LIN {X 0,Y 257.253,Z 513.083,A -85,B 0,C 180,E1 -18787.513,E2 -18787.513} C_VEL
LIN {X 0,Y 254.562,Z 521.781,A -85,B 0,C 180,E1 -18789.728,E2 -18789.728} C_VEL
LIN {X 0,Y 252.293,Z 529.293,A -85,B 0,C 180,E1 -18792.156,E2 -18792.156} C_VEL
LIN {X 0,Y 250.394,Z 535.119,A -85,B 0,C 180,E1 -18794.535,E2 -18794.535} C_VEL
LIN {X 0,Y 248.86,Z 539.729,A -85,B 0,C 180,E1 -18796.942,E2 -18796.942} C_VEL
LIN {X 0,Y 247.896,Z 543.258,A -85,B 0,C 180,E1 -18799.38,E2 -18799.38} C_VEL
LIN {X 0,Y 247.266,Z 545.801,A -85,B 0,C 180,E1 -18801.829,E2 -18801.829} C_VEL
LIN {X 0,Y 247.011,Z 547.002,A -85,B 0,C 180,E1 -18803.465,E2 -18803.465} C_VEL
LIN {X 0,Y 246.916,Z 548.152,A -85,B 0,C 180,E1 -18806.736,E2 -18806.736} C_VEL
LIN {X 0,Y 246.997,Z 548.151,A -85,B 0,C 180,E1 -18808.369,E2 -18808.369} C_VEL
LIN {X 0,Y 247.028,Z 547.759,A -85,B 0,C 180,E1 -18809.999,E2 -18809.999} C_VEL
LIN {X 0,Y 247.02,Z 546.926,A -85,B 0,C 180,E1 -18811.63,E2 -18811.63} C_VEL
LIN {X 0,Y 246.98,Z 545.678,A -85,B 0,C 180,E1 -18813.262,E2 -18813.262} C_VEL
LIN {X 0,Y 246.984,Z 543.722,A -85,B 0,C 180,E1 -18815.163,E2 -18815.163} C_VEL
LIN {X 0,Y 247.156,Z 540.666,A -85,B 0,C 180,E1 -18817.351,E2 -18817.351} C_VEL
LIN {X 0,Y 247.53,Z 536.217,A -85,B 0,C 180,E1 -18819.808,E2 -18819.808} C_VEL
LIN {X 0,Y 248.187,Z 530.545,A -85,B 0,C 180,E1 -18822.261,E2 -18822.261} C_VEL
LIN {X 0,Y 249.393,Z 523.451,A -85,B 0,C 180,E1 -18824.691,E2 -18824.691} C_VEL
LIN {X 0,Y 250.655,Z 516.203,A -85,B 0,C 180,E1 -18826.701,E2 -18826.701} C_VEL
LIN {X 0,Y 252.124,Z 506.524,A -85,B 0,C 180,E1 -18828.879,E2 -18828.879} C_VEL
LIN {X 0,Y 253.731,Z 496.53,A -85,B 0,C 180,E1 -18830.68,E2 -18830.68} C_VEL
LIN {X 0,Y 255.423,Z 485.697,A -85,B 0,C 180,E1 -18832.23,E2 -18832.23} C_VEL
LIN {X 0,Y 257.066,Z 473.51,A -85,B 0,C 180,E1 -18833.567,E2 -18833.567} C_VEL
LIN {X 0,Y 258.522,Z 460.783,A -85,B 0,C 180,E1 -18834.599,E2 -18834.599} C_VEL
LIN {X 0,Y 259.525,Z 448.241,A -85,B 0,C 180,E1 -18835.299,E2 -18835.299} C_VEL
LIN {X 0,Y 260.096,Z 431.393,A -85,B 0,C 180,E1 -18835.851,E2 -18835.851} C_VEL
LIN {X 0,Y 261.403,Z 385.497,A -85,B 0,C 180,E1 -18837.079,E2 -18837.079} C_VEL
LIN {X 0,Y 257.137,Z 350.583,A -85,B 0,C 180,E1 -18838.529,E2 -18838.529} C_VEL
LIN {X 0,Y 256.159,Z 345.324,A -85,B 0,C 180,E1 -18838.787,E2 -18838.787} C_VEL
LIN {X 0,Y 252.427,Z 335.153,A -85,B 0,C 180,E1 -18839.536,E2 -18839.536} C_VEL
LIN {X 0,Y 250.251,Z 324.745,A -85,B 0,C 180,E1 -18843.339,E2 -18843.339} C_VEL
LIN {X 0,Y 249.089,Z 319.458,A -85,B 0,C 180,E1 -18845.38,E2 -18845.38} C_VEL
LIN {X 0,Y 249.027,Z 319.467,A -85,B 0,C 180,E1 -18848.379,E2 -18848.379} C_VEL
LIN {X 0,Y 249,Z 319.469,A -85,B 0,C 180,E1 -18852.79,E2 -18852.79} C_VEL
LIN {X 0,Y 249.008,Z 319.467,A -85,B 0,C 180,E1 -18857.361,E2 -18857.361} C_VEL
LIN {X 0,Y 249.024,Z 319.466,A -85,B 0,C 180,E1 -18861.618,E2 -18861.618} C_VEL
LIN {X 0,Y 249.041,Z 319.463,A -85,B 0,C 180,E1 -18865.639,E2 -18865.639} C_VEL
LIN {X 0,Y 249.049,Z 319.463,A -85,B 0,C 180,E1 -18869.472,E2 -18869.472} C_VEL
LIN {X 0,Y 249.07,Z 319.462,A -85,B 0,C 180,E1 -18873.161,E2 -18873.161} C_VEL
LIN {X 0,Y 249.076,Z 319.46,A -85,B 0,C 180,E1 -18876.732,E2 -18876.732} C_VEL
LIN {X 0,Y 249.108,Z 319.453,A -85,B 0,C 180,E1 -18880.211,E2 -18880.211} C_VEL
LIN {X 0,Y 249.239,Z 319.439,A -85,B 0,C 180,E1 -18883.621,E2 -18883.621} C_VEL
LIN {X 0,Y 249.249,Z 319.422,A -85,B 0,C 180,E1 -18888.616,E2 -18888.616} C_VEL
LIN {X 0,Y 249.476,Z 319.408,A -85,B 0,C 180,E1 -18891.902,E2 -18891.902} C_VEL
LIN {X 0,Y 249.43,Z 319.409,A -85,B 0,C 180,E1 -18896.769,E2 -18896.769} C_VEL
LIN {X 0,Y 249.717,Z 319.366,A -85,B 0,C 180,E1 -18900,E2 -18900} C_VEL
LIN {X 0,Y 249.428,Z 319.412,A -85,B 0,C 180,E1 -18903.23,E2 -18903.23} C_VEL
LIN {X 0,Y 249.428,Z 319.41,A -85,B 0,C 180,E1 -18906.548,E2 -18906.548} C_VEL
LIN {X 0,Y 249.339,Z 319.412,A -85,B 0,C 180,E1 -18909.736,E2 -18909.736} C_VEL
LIN {X 0,Y 249.201,Z 319.442,A -85,B 0,C 180,E1 -18914.703,E2 -18914.703} C_VEL
LIN {X 0,Y 249.134,Z 319.446,A -85,B 0,C 180,E1 -18918.077,E2 -18918.077} C_VEL
LIN {X 0,Y 249.08,Z 319.446,A -85,B 0,C 180,E1 -18921.518,E2 -18921.518} C_VEL
LIN {X 0,Y 249.113,Z 319.452,A -85,B 0,C 180,E1 -18925.476,E2 -18925.476} C_VEL
LIN {X 0,Y 249.079,Z 319.446,A -85,B 0,C 180,E1 -18928.994,E2 -18928.994} C_VEL
LIN {X 0,Y 249.027,Z 319.459,A -85,B 0,C 180,E1 -18932.426,E2 -18932.426} C_VEL
LIN {X 0,Y 249.043,Z 319.461,A -85,B 0,C 180,E1 -18936.343,E2 -18936.343} C_VEL
LIN {X 0,Y 249.002,Z 319.461,A -85,B 0,C 180,E1 -18940.478,E2 -18940.478} C_VEL
LIN {X 0,Y 248.998,Z 319.469,A -85,B 0,C 180,E1 -18942.791,E2 -18942.791} C_VEL
LIN {X 0,Y 248.977,Z 319.469,A -85,B 0,C 180,E1 -18947.356,E2 -18947.356} C_VEL
LIN {X 0,Y 249.038,Z 319.457,A -85,B 0,C 180,E1 -18952.201,E2 -18952.201} C_VEL
LIN {X 0,Y 249.04,Z 319.463,A -85,B 0,C 180,E1 -18955.64,E2 -18955.64} C_VEL
LIN {X 0,Y 248.991,Z 319.466,A -85,B 0,C 180,E1 -18959.466,E2 -18959.466} C_VEL
LIN {X 0,Y 249.014,Z 319.463,A -85,B 0,C 180,E1 -18963.156,E2 -18963.156} C_VEL
LIN {X 0,Y 249.018,Z 319.465,A -85,B 0,C 180,E1 -18966.727,E2 -18966.727} C_VEL
LIN {X 0,Y 249.107,Z 319.48,A -85,B 0,C 180,E1 -18970.25,E2 -18970.25} C_VEL
LIN {X 0,Y 250.158,Z 322.4,A -85,B 0,C 180,E1 -18970.459,E2 -18970.459} C_VEL
LIN {X 0,Y 254.562,Z 332.022,A -85,B 0,C 180,E1 -18971.233,E2 -18971.233} C_VEL
LIN {X 0,Y 261.497,Z 350.837,A -85,B 0,C 180,E1 -18972.499,E2 -18972.499} C_VEL
LIN {X 0,Y 262.283,Z 353.529,A -85,B 0,C 180,E1 -18972.654,E2 -18972.654} C_VEL
LIN {X 0,Y 260.108,Z 426.14,A -85,B 0,C 180,E1 -18974.626,E2 -18974.626} C_VEL
LIN {X 0,Y 259.371,Z 439.258,A -85,B 0,C 180,E1 -18975.285,E2 -18975.285} C_VEL
LIN {X 0,Y 258.324,Z 451.887,A -85,B 0,C 180,E1 -18976.229,E2 -18976.229} C_VEL
LIN {X 0,Y 257.112,Z 463.144,A -85,B 0,C 180,E1 -18977.369,E2 -18977.369} C_VEL
LIN {X 0,Y 255.161,Z 474.833,A -85,B 0,C 180,E1 -18978.884,E2 -18978.884} C_VEL
LIN {X 0,Y 253.619,Z 485.254,A -85,B 0,C 180,E1 -18980.631,E2 -18980.631} C_VEL
LIN {X 0,Y 252.118,Z 493.801,A -85,B 0,C 180,E1 -18982.392,E2 -18982.392} C_VEL
LIN {X 0,Y 250.826,Z 501.662,A -85,B 0,C 180,E1 -18984.373,E2 -18984.373} C_VEL
LIN {X 0,Y 249.426,Z 509.37,A -85,B 0,C 180,E1 -18986.77,E2 -18986.77} C_VEL
LIN {X 0,Y 248.464,Z 515.541,A -85,B 0,C 180,E1 -18989.19,E2 -18989.19} C_VEL
LIN {X 0,Y 247.694,Z 520.458,A -85,B 0,C 180,E1 -18991.626,E2 -18991.626} C_VEL
LIN {X 0,Y 247.377,Z 524.246,A -85,B 0,C 180,E1 -18994.073,E2 -18994.073} C_VEL
LIN {X 0,Y 247.112,Z 527.029,A -85,B 0,C 180,E1 -18996.533,E2 -18996.533} C_VEL
LIN {X 0,Y 246.903,Z 528.355,A -85,B 0,C 180,E1 -18998.183,E2 -18998.183} C_VEL
LIN {X 0,Y 246.8,Z 529.286,A -85,B 0,C 180,E1 -18999.838,E2 -18999.838} C_VEL
LIN {X 0,Y 246.83,Z 529.798,A -85,B 0,C 180,E1 -19001.497,E2 -19001.497} C_VEL
LIN {X 0,Y 247.025,Z 529.882,A -85,B 0,C 180,E1 -19003.157,E2 -19003.157} C_VEL
LIN {X 0,Y 247.338,Z 529.537,A -85,B 0,C 180,E1 -19004.964,E2 -19004.964} C_VEL
LIN {X 0,Y 247.629,Z 528.884,A -85,B 0,C 180,E1 -19006.488,E2 -19006.488} C_VEL
LIN {X 0,Y 248.082,Z 527.744,A -85,B 0,C 180,E1 -19008.158,E2 -19008.158} C_VEL
LIN {X 0,Y 249.053,Z 525.234,A -85,B 0,C 180,E1 -19010.655,E2 -19010.655} C_VEL
LIN {X 0,Y 250.39,Z 521.674,A -85,B 0,C 180,E1 -19013.139,E2 -19013.139} C_VEL
LIN {X 0,Y 252.11,Z 516.953,A -85,B 0,C 180,E1 -19015.601,E2 -19015.601} C_VEL
LIN {X 0,Y 254.147,Z 510.919,A -85,B 0,C 180,E1 -19018.041,E2 -19018.041} C_VEL
LIN {X 0,Y 256.653,Z 503.353,A -85,B 0,C 180,E1 -19020.437,E2 -19020.437} C_VEL
LIN {X 0,Y 259.061,Z 495.585,A -85,B 0,C 180,E1 -19022.398,E2 -19022.398} C_VEL
LIN {X 0,Y 261.749,Z 486.067,A -85,B 0,C 180,E1 -19024.323,E2 -19024.323} C_VEL
LIN {X 0,Y 264.345,Z 475.395,A -85,B 0,C 180,E1 -19026.032,E2 -19026.032} C_VEL
LIN {X 0,Y 266.477,Z 465.074,A -85,B 0,C 180,E1 -19027.344,E2 -19027.344} C_VEL
LIN {X 0,Y 268.474,Z 453.071,A -85,B 0,C 180,E1 -19028.536,E2 -19028.536} C_VEL
LIN {X 0,Y 269.983,Z 440.573,A -85,B 0,C 180,E1 -19029.444,E2 -19029.444} C_VEL
LIN {X 0,Y 270.997,Z 428.372,A -85,B 0,C 180,E1 -19030.052,E2 -19030.052} C_VEL
LIN {X 0,Y 272.213,Z 404.536,A -85,B 0,C 180,E1 -19030.702,E2 -19030.702} C_VEL
LIN {X 0,Y 273.903,Z 366.243,A -85,B 0,C 180,E1 -19031.667,E2 -19031.667} C_VEL
LIN {X 0,Y 267.043,Z 351.29,A -85,B 0,C 180,E1 -19033.238,E2 -19033.238} C_VEL
LIN {X 0,Y 260.131,Z 338.414,A -85,B 0,C 180,E1 -19034.869,E2 -19034.869} C_VEL
LIN {X 0,Y 253.898,Z 327.876,A -85,B 0,C 180,E1 -19036.414,E2 -19036.414} C_VEL
LIN {X 0,Y 251.287,Z 323.854,A -85,B 0,C 180,E1 -19037.081,E2 -19037.081} C_VEL
LIN {X 0,Y 249.658,Z 321.603,A -85,B 0,C 180,E1 -19037.499,E2 -19037.499} C_VEL
LIN {X 0,Y 249.109,Z 319.866,A -85,B 0,C 180,E1 -19037.725,E2 -19037.725} C_VEL
LIN {X 0,Y 249.017,Z 319.466,A -85,B 0,C 180,E1 -19038.047,E2 -19038.047} C_VEL
LIN {X 0,Y 249.043,Z 319.458,A -85,B 0,C 180,E1 -19042.201,E2 -19042.201} C_VEL
LIN {X 0,Y 249.044,Z 319.457,A -85,B 0,C 180,E1 -19045.64,E2 -19045.64} C_VEL
LIN {X 0,Y 249.052,Z 319.447,A -85,B 0,C 180,E1 -19049.474,E2 -19049.474} C_VEL
LIN {X 0,Y 249.07,Z 319.445,A -85,B 0,C 180,E1 -19053.162,E2 -19053.162} C_VEL
LIN {X 0,Y 249.062,Z 319.446,A -85,B 0,C 180,E1 -19056.731,E2 -19056.731} C_VEL
LIN {X 0,Y 249.108,Z 319.442,A -85,B 0,C 180,E1 -19060.212,E2 -19060.212} C_VEL
LIN {X 0,Y 249.243,Z 319.433,A -85,B 0,C 180,E1 -19063.622,E2 -19063.622} C_VEL
LIN {X 0,Y 249.254,Z 319.428,A -85,B 0,C 180,E1 -19068.617,E2 -19068.617} C_VEL
LIN {X 0,Y 249.485,Z 319.406,A -85,B 0,C 180,E1 -19071.903,E2 -19071.903} C_VEL
LIN {X 0,Y 249.436,Z 319.409,A -85,B 0,C 180,E1 -19076.77,E2 -19076.77} C_VEL
LIN {X 0,Y 249.722,Z 319.376,A -85,B 0,C 180,E1 -19080,E2 -19080} C_VEL
LIN {X 0,Y 249.643,Z 319.378,A -85,B 0,C 180,E1 -19081.777,E2 -19081.777} C_VEL
LIN {X 0,Y 248.799,Z 319.482,A -85,B 0,C 180,E1 -19083.121,E2 -19083.121} C_VEL
LIN {X 0,Y 245.894,Z 319.852,A -85,B 0,C 180,E1 -19085.314,E2 -19085.314} C_VEL
LIN {X 0,Y 243.517,Z 320.143,A -85,B 0,C 180,E1 -19087.099,E2 -19087.099} C_VEL
LIN {X 0,Y 242.483,Z 320.272,A -85,B 0,C 180,E1 -19088.482,E2 -19088.482} C_VEL
LIN {X 0,Y 242.384,Z 320.284,A -85,B 0,C 180,E1 -19088.951,E2 -19088.951} C_VEL
LIN {X 0,Y 242.168,Z 320.316,A -85,B 0,C 180,E1 -19093.425,E2 -19093.425} C_VEL
LIN {X 0,Y 242.152,Z 320.311,A -85,B 0,C 180,E1 -19096.872,E2 -19096.872} C_VEL
LIN {X 0,Y 242.028,Z 320.333,A -85,B 0,C 180,E1 -19101.687,E2 -19101.687} C_VEL
LIN {X 0,Y 242.069,Z 320.328,A -85,B 0,C 180,E1 -19105.838,E2 -19105.838} C_VEL
LIN {X 0,Y 242.009,Z 320.334,A -85,B 0,C 180,E1 -19109.583,E2 -19109.583} C_VEL
LIN {X 0,Y 241.983,Z 320.338,A -85,B 0,C 180,E1 -19113.493,E2 -19113.493} C_VEL
LIN {X 0,Y 241.989,Z 320.341,A -85,B 0,C 180,E1 -19117.582,E2 -19117.582} C_VEL
LIN {X 0,Y 241.932,Z 320.329,A -85,B 0,C 180,E1 -19121.924,E2 -19121.924} C_VEL
LIN {X 0,Y 241.986,Z 320.464,A -85,B 0,C 180,E1 -19125.087,E2 -19125.087} C_VEL
LIN {X 0,Y 244.554,Z 329.275,A -85,B 0,C 180,E1 -19129.602,E2 -19129.602} C_VEL
LIN {X 0,Y 245.765,Z 333.657,A -85,B 0,C 180,E1 -19131.684,E2 -19131.684} C_VEL
LIN {X 0,Y 248.353,Z 338.358,A -85,B 0,C 180,E1 -19132.407,E2 -19132.407} C_VEL
LIN {X 0,Y 256.334,Z 353.521,A -85,B 0,C 180,E1 -19134.512,E2 -19134.512} C_VEL
LIN {X 0,Y 262.927,Z 367.737,A -85,B 0,C 180,E1 -19136.166,E2 -19136.166} C_VEL
LIN {X 0,Y 264.065,Z 371.108,A -85,B 0,C 180,E1 -19136.47,E2 -19136.47} C_VEL
LIN {X 0,Y 267.144,Z 390.198,A -85,B 0,C 180,E1 -19137.602,E2 -19137.602} C_VEL
LIN {X 0,Y 264.881,Z 443.227,A -85,B 0,C 180,E1 -19139.029,E2 -19139.029} C_VEL
LIN {X 0,Y 263.521,Z 456.86,A -85,B 0,C 180,E1 -19139.665,E2 -19139.665} C_VEL
LIN {X 0,Y 261.592,Z 469.409,A -85,B 0,C 180,E1 -19140.528,E2 -19140.528} C_VEL
LIN {X 0,Y 259.274,Z 481.377,A -85,B 0,C 180,E1 -19141.682,E2 -19141.682} C_VEL
LIN {X 0,Y 256.566,Z 492.822,A -85,B 0,C 180,E1 -19143.129,E2 -19143.129} C_VEL
LIN {X 0,Y 253.805,Z 503.151,A -85,B 0,C 180,E1 -19144.802,E2 -19144.802} C_VEL
LIN {X 0,Y 251.249,Z 511.614,A -85,B 0,C 180,E1 -19146.509,E2 -19146.509} C_VEL
LIN {X 0,Y 248.707,Z 519.442,A -85,B 0,C 180,E1 -19148.447,E2 -19148.447} C_VEL
LIN {X 0,Y 246.267,Z 527.109,A -85,B 0,C 180,E1 -19150.841,E2 -19150.841} C_VEL
LIN {X 0,Y 244.208,Z 533.294,A -85,B 0,C 180,E1 -19153.274,E2 -19153.274} C_VEL
LIN {X 0,Y 242.408,Z 538.231,A -85,B 0,C 180,E1 -19155.733,E2 -19155.733} C_VEL
LIN {X 0,Y 241.211,Z 542.064,A -85,B 0,C 180,E1 -19158.231,E2 -19158.231} C_VEL
LIN {X 0,Y 240.216,Z 545.635,A -85,B 0,C 180,E1 -19161.588,E2 -19161.588} C_VEL
LIN {X 0,Y 239.953,Z 546.795,A -85,B 0,C 180,E1 -19163.271,E2 -19163.271} C_VEL
LIN {X 0,Y 239.816,Z 547.898,A -85,B 0,C 180,E1 -19166.639,E2 -19166.639} C_VEL
LIN {X 0,Y 239.903,Z 547.876,A -85,B 0,C 180,E1 -19168.321,E2 -19168.321} C_VEL
LIN {X 0,Y 239.957,Z 547.451,A -85,B 0,C 180,E1 -19169.999,E2 -19169.999} C_VEL
LIN {X 0,Y 239.927,Z 546.584,A -85,B 0,C 180,E1 -19171.678,E2 -19171.678} C_VEL
LIN {X 0,Y 239.879,Z 545.313,A -85,B 0,C 180,E1 -19173.359,E2 -19173.359} C_VEL
LIN {X 0,Y 239.919,Z 542.599,A -85,B 0,C 180,E1 -19175.884,E2 -19175.884} C_VEL
LIN {X 0,Y 240.178,Z 538.844,A -85,B 0,C 180,E1 -19178.412,E2 -19178.412} C_VEL
LIN {X 0,Y 240.703,Z 533.946,A -85,B 0,C 180,E1 -19180.94,E2 -19180.94} C_VEL
LIN {X 0,Y 241.585,Z 527.758,A -85,B 0,C 180,E1 -19183.457,E2 -19183.457} C_VEL
LIN {X 0,Y 242.909,Z 520.055,A -85,B 0,C 180,E1 -19185.953,E2 -19185.953} C_VEL
LIN {X 0,Y 244.376,Z 512.158,A -85,B 0,C 180,E1 -19188.008,E2 -19188.008} C_VEL
LIN {X 0,Y 245.855,Z 502.462,A -85,B 0,C 180,E1 -19190.061,E2 -19190.061} C_VEL
LIN {X 0,Y 247.707,Z 491.733,A -85,B 0,C 180,E1 -19191.862,E2 -19191.862} C_VEL
LIN {X 0,Y 249.32,Z 481.357,A -85,B 0,C 180,E1 -19193.243,E2 -19193.243} C_VEL
LIN {X 0,Y 250.912,Z 468.939,A -85,B 0,C 180,E1 -19194.512,E2 -19194.512} C_VEL
LIN {X 0,Y 252.312,Z 455.866,A -85,B 0,C 180,E1 -19195.467,E2 -19195.467} C_VEL
LIN {X 0,Y 253.19,Z 443.052,A -85,B 0,C 180,E1 -19196.089,E2 -19196.089} C_VEL
LIN {X 0,Y 254.817,Z 385.79,A -85,B 0,C 180,E1 -19197.694,E2 -19197.694} C_VEL
LIN {X 0,Y 250.723,Z 351.896,A -85,B 0,C 180,E1 -19199.15,E2 -19199.15} C_VEL
LIN {X 0,Y 249.794,Z 347.296,A -85,B 0,C 180,E1 -19199.392,E2 -19199.392} C_VEL
LIN {X 0,Y 245.198,Z 334.962,A -85,B 0,C 180,E1 -19200.308,E2 -19200.308} C_VEL
LIN {X 0,Y 242.927,Z 324.358,A -85,B 0,C 180,E1 -19204.342,E2 -19204.342} C_VEL
LIN {X 0,Y 242.051,Z 320.334,A -85,B 0,C 180,E1 -19206.01,E2 -19206.01} C_VEL
LIN {X 0,Y 241.956,Z 320.346,A -85,B 0,C 180,E1 -19209.718,E2 -19209.718} C_VEL
LIN {X 0,Y 241.917,Z 320.352,A -85,B 0,C 180,E1 -19214.204,E2 -19214.204} C_VEL
LIN {X 0,Y 241.932,Z 320.349,A -85,B 0,C 180,E1 -19218.076,E2 -19218.076} C_VEL
LIN {X 0,Y 241.984,Z 320.344,A -85,B 0,C 180,E1 -19222.417,E2 -19222.417} C_VEL
LIN {X 0,Y 241.978,Z 320.345,A -85,B 0,C 180,E1 -19226.507,E2 -19226.507} C_VEL
LIN {X 0,Y 242.034,Z 320.339,A -85,B 0,C 180,E1 -19230.586,E2 -19230.586} C_VEL
LIN {X 0,Y 242.065,Z 320.331,A -85,B 0,C 180,E1 -19234.182,E2 -19234.182} C_VEL
LIN {X 0,Y 242.05,Z 320.331,A -85,B 0,C 180,E1 -19238.296,E2 -19238.296} C_VEL
LIN {X 0,Y 242.16,Z 320.322,A -85,B 0,C 180,E1 -19243.278,E2 -19243.278} C_VEL
LIN {X 0,Y 242.183,Z 320.301,A -85,B 0,C 180,E1 -19248.279,E2 -19248.279} C_VEL
LIN {X 0,Y 242.423,Z 320.284,A -85,B 0,C 180,E1 -19251.665,E2 -19251.665} C_VEL
LIN {X 0,Y 242.254,Z 320.307,A -85,B 0,C 180,E1 -19255.007,E2 -19255.007} C_VEL
LIN {X 0,Y 242.632,Z 320.246,A -85,B 0,C 180,E1 -19258.34,E2 -19258.34} C_VEL
LIN {X 0,Y 242.631,Z 320.254,A -85,B 0,C 180,E1 -19261.659,E2 -19261.659} C_VEL
LIN {X 0,Y 242.404,Z 320.285,A -85,B 0,C 180,E1 -19266.659,E2 -19266.659} C_VEL
LIN {X 0,Y 242.263,Z 320.292,A -85,B 0,C 180,E1 -19270.024,E2 -19270.024} C_VEL
LIN {X 0,Y 242.163,Z 320.318,A -85,B 0,C 180,E1 -19275.141,E2 -19275.141} C_VEL
LIN {X 0,Y 242.067,Z 320.321,A -85,B 0,C 180,E1 -19278.624,E2 -19278.624} C_VEL
LIN {X 0,Y 242.002,Z 320.331,A -85,B 0,C 180,E1 -19282.181,E2 -19282.181} C_VEL
LIN {X 0,Y 242.063,Z 320.331,A -85,B 0,C 180,E1 -19285.838,E2 -19285.838} C_VEL
LIN {X 0,Y 242.026,Z 320.323,A -85,B 0,C 180,E1 -19289.58,E2 -19289.58} C_VEL
LIN {X 0,Y 241.977,Z 320.34,A -85,B 0,C 180,E1 -19293.493,E2 -19293.493} C_VEL
LIN {X 0,Y 241.985,Z 320.332,A -85,B 0,C 180,E1 -19297.582,E2 -19297.582} C_VEL
LIN {X 0,Y 241.93,Z 320.346,A -85,B 0,C 180,E1 -19301.924,E2 -19301.924} C_VEL
LIN {X 0,Y 241.901,Z 320.342,A -85,B 0,C 180,E1 -19306.579,E2 -19306.579} C_VEL
LIN {X 0,Y 241.99,Z 320.335,A -85,B 0,C 180,E1 -19311.642,E2 -19311.642} C_VEL
LIN {X 0,Y 241.984,Z 320.341,A -85,B 0,C 180,E1 -19314.49,E2 -19314.49} C_VEL
LIN {X 0,Y 241.945,Z 320.345,A -85,B 0,C 180,E1 -19318.477,E2 -19318.477} C_VEL
LIN {X 0,Y 241.95,Z 320.342,A -85,B 0,C 180,E1 -19322.306,E2 -19322.306} C_VEL
LIN {X 0,Y 241.991,Z 320.341,A -85,B 0,C 180,E1 -19326.01,E2 -19326.01} C_VEL
LIN {X 0,Y 242.018,Z 320.339,A -85,B 0,C 180,E1 -19329.426,E2 -19329.426} C_VEL
LIN {X 0,Y 243.035,Z 323.201,A -85,B 0,C 180,E1 -19329.669,E2 -19329.669} C_VEL
LIN {X 0,Y 247.68,Z 332.843,A -85,B 0,C 180,E1 -19330.512,E2 -19330.512} C_VEL
LIN {X 0,Y 254.536,Z 350.896,A -85,B 0,C 180,E1 -19331.808,E2 -19331.808} C_VEL
LIN {X 0,Y 255.778,Z 354.774,A -85,B 0,C 180,E1 -19332.052,E2 -19332.052} C_VEL
LIN {X 0,Y 253.504,Z 426.848,A -85,B 0,C 180,E1 -19334.06,E2 -19334.06} C_VEL
LIN {X 0,Y 252.689,Z 440.569,A -85,B 0,C 180,E1 -19334.783,E2 -19334.783} C_VEL
LIN {X 0,Y 251.612,Z 452.915,A -85,B 0,C 180,E1 -19335.751,E2 -19335.751} C_VEL
LIN {X 0,Y 250.262,Z 464.743,A -85,B 0,C 180,E1 -19337.018,E2 -19337.018} C_VEL
LIN {X 0,Y 248.442,Z 474.903,A -85,B 0,C 180,E1 -19338.373,E2 -19338.373} C_VEL
LIN {X 0,Y 246.826,Z 485.36,A -85,B 0,C 180,E1 -19340.164,E2 -19340.164} C_VEL
LIN {X 0,Y 245.114,Z 494.815,A -85,B 0,C 180,E1 -19342.173,E2 -19342.173} C_VEL
LIN {X 0,Y 243.538,Z 503.893,A -85,B 0,C 180,E1 -19344.619,E2 -19344.619} C_VEL
LIN {X 0,Y 242.134,Z 511.228,A -85,B 0,C 180,E1 -19347.089,E2 -19347.089} C_VEL
LIN {X 0,Y 241.11,Z 517.947,A -85,B 0,C 180,E1 -19350.001,E2 -19350.001} C_VEL
LIN {X 0,Y 240.426,Z 522.397,A -85,B 0,C 180,E1 -19352.514,E2 -19352.514} C_VEL
LIN {X 0,Y 240.18,Z 525.767,A -85,B 0,C 180,E1 -19355.037,E2 -19355.037} C_VEL
LIN {X 0,Y 239.982,Z 527.454,A -85,B 0,C 180,E1 -19356.728,E2 -19356.728} C_VEL
LIN {X 0,Y 239.792,Z 528.744,A -85,B 0,C 180,E1 -19358.427,E2 -19358.427} C_VEL
LIN {X 0,Y 239.723,Z 529.635,A -85,B 0,C 180,E1 -19360.132,E2 -19360.132} C_VEL
LIN {X 0,Y 239.776,Z 530.083,A -85,B 0,C 180,E1 -19361.84,E2 -19361.84} C_VEL
LIN {X 0,Y 240.309,Z 529.794,A -85,B 0,C 180,E1 -19365.261,E2 -19365.261} C_VEL
LIN {X 0,Y 240.648,Z 529.054,A -85,B 0,C 180,E1 -19366.981,E2 -19366.981} C_VEL
LIN {X 0,Y 241.152,Z 527.856,A -85,B 0,C 180,E1 -19368.698,E2 -19368.698} C_VEL
LIN {X 0,Y 241.845,Z 526.242,A -85,B 0,C 180,E1 -19370.409,E2 -19370.409} C_VEL
LIN {X 0,Y 243.163,Z 522.965,A -85,B 0,C 180,E1 -19372.966,E2 -19372.966} C_VEL
LIN {X 0,Y 244.862,Z 518.568,A -85,B 0,C 180,E1 -19375.501,E2 -19375.501} C_VEL
LIN {X 0,Y 247.006,Z 512.67,A -85,B 0,C 180,E1 -19378.112,E2 -19378.112} C_VEL
LIN {X 0,Y 249.444,Z 505.79,A -85,B 0,C 180,E1 -19380.474,E2 -19380.474} C_VEL
LIN {X 0,Y 252.406,Z 496.805,A -85,B 0,C 180,E1 -19382.886,E2 -19382.886} C_VEL
LIN {X 0,Y 255.171,Z 487.541,A -85,B 0,C 180,E1 -19384.855,E2 -19384.855} C_VEL
LIN {X 0,Y 257.856,Z 477.179,A -85,B 0,C 180,E1 -19386.6,E2 -19386.6} C_VEL
LIN {X 0,Y 260.392,Z 465.583,A -85,B 0,C 180,E1 -19388.127,E2 -19388.127} C_VEL
LIN {X 0,Y 262.492,Z 453.54,A -85,B 0,C 180,E1 -19389.349,E2 -19389.349} C_VEL
LIN {X 0,Y 264.13,Z 440.525,A -85,B 0,C 180,E1 -19390.309,E2 -19390.309} C_VEL
LIN {X 0,Y 265.185,Z 428.167,A -85,B 0,C 180,E1 -19390.928,E2 -19390.928} C_VEL
LIN {X 0,Y 266.582,Z 400.796,A -85,B 0,C 180,E1 -19391.674,E2 -19391.674} C_VEL
LIN {X 0,Y 268.012,Z 368.143,A -85,B 0,C 180,E1 -19392.521,E2 -19392.521} C_VEL
LIN {X 0,Y 260.943,Z 352.931,A -85,B 0,C 180,E1 -19394.219,E2 -19394.219} C_VEL
LIN {X 0,Y 254.159,Z 340.365,A -85,B 0,C 180,E1 -19395.906,E2 -19395.906} C_VEL
LIN {X 0,Y 249.492,Z 332.557,A -85,B 0,C 180,E1 -19397.116,E2 -19397.116} C_VEL
LIN {X 0,Y 246.884,Z 328.628,A -85,B 0,C 180,E1 -19397.807,E2 -19397.807} C_VEL
LIN {X 0,Y 244.466,Z 324.912,A -85,B 0,C 180,E1 -19398.471,E2 -19398.471} C_VEL
LIN {X 0,Y 242.615,Z 322.568,A -85,B 0,C 180,E1 -19398.974,E2 -19398.974} C_VEL
LIN {X 0,Y 241.977,Z 320.342,A -85,B 0,C 180,E1 -19399.252,E2 -19399.252} C_VEL
LIN {X 0,Y 241.989,Z 320.338,A -85,B 0,C 180,E1 -19402.418,E2 -19402.418} C_VEL
LIN {X 0,Y 241.981,Z 320.334,A -85,B 0,C 180,E1 -19406.508,E2 -19406.508} C_VEL
LIN {X 0,Y 242.037,Z 320.327,A -85,B 0,C 180,E1 -19410.588,E2 -19410.588} C_VEL
LIN {X 0,Y 242.068,Z 320.325,A -85,B 0,C 180,E1 -19414.183,E2 -19414.183} C_VEL
LIN {X 0,Y 242.027,Z 320.333,A -85,B 0,C 180,E1 -19418.314,E2 -19418.314} C_VEL
LIN {X 0,Y 242.164,Z 320.318,A -85,B 0,C 180,E1 -19423.279,E2 -19423.279} C_VEL
LIN {X 0,Y 242.187,Z 320.31,A -85,B 0,C 180,E1 -19428.28,E2 -19428.28} C_VEL
LIN {X 0,Y 242.436,Z 320.286,A -85,B 0,C 180,E1 -19431.666,E2 -19431.666} C_VEL
LIN {X 0,Y 242.26,Z 320.304,A -85,B 0,C 180,E1 -19435.008,E2 -19435.008} C_VEL
LIN {X 0,Y 242.637,Z 320.249,A -85,B 0,C 180,E1 -19438.341,E2 -19438.341} C_VEL
LIN {X 0,Y 242.629,Z 320.252,A -85,B 0,C 180,E1 -19441.694,E2 -19441.694} C_VEL
LIN {X 0,Y 242.434,Z 320.272,A -85,B 0,C 180,E1 -19446.659,E2 -19446.659} C_VEL
LIN {X 0,Y 242.384,Z 320.284,A -85,B 0,C 180,E1 -19448.951,E2 -19448.951} C_VEL
LIN {X 0,Y 241.655,Z 320.381,A -85,B 0,C 180,E1 -19450.336,E2 -19450.336} C_VEL
LIN {X 0,Y 238.711,Z 320.744,A -85,B 0,C 180,E1 -19452.593,E2 -19452.593} C_VEL
LIN {X 0,Y 236.236,Z 321.055,A -85,B 0,C 180,E1 -19454.431,E2 -19454.431} C_VEL
LIN {X 0,Y 235.176,Z 321.178,A -85,B 0,C 180,E1 -19455.861,E2 -19455.861} C_VEL
LIN {X 0,Y 235.09,Z 321.188,A -85,B 0,C 180,E1 -19456.345,E2 -19456.345} C_VEL
LIN {X 0,Y 235,Z 321.202,A -85,B 0,C 180,E1 -19461.032,E2 -19461.032} C_VEL
LIN {X 0,Y 234.996,Z 321.211,A -85,B 0,C 180,E1 -19466.206,E2 -19466.206} C_VEL
LIN {X 0,Y 234.924,Z 321.223,A -85,B 0,C 180,E1 -19470.569,E2 -19470.569} C_VEL
LIN {X 0,Y 234.929,Z 321.219,A -85,B 0,C 180,E1 -19474.639,E2 -19474.639} C_VEL
LIN {X 0,Y 234.915,Z 321.204,A -85,B 0,C 180,E1 -19478.936,E2 -19478.936} C_VEL
LIN {X 0,Y 234.899,Z 321.306,A -85,B 0,C 180,E1 -19483.661,E2 -19483.661} C_VEL
LIN {X 0,Y 237.521,Z 330.019,A -85,B 0,C 180,E1 -19488.403,E2 -19488.403} C_VEL
LIN {X 0,Y 238.489,Z 333.51,A -85,B 0,C 180,E1 -19490.066,E2 -19490.066} C_VEL
LIN {X 0,Y 240.919,Z 337.776,A -85,B 0,C 180,E1 -19490.795,E2 -19490.795} C_VEL
LIN {X 0,Y 245.507,Z 345.979,A -85,B 0,C 180,E1 -19492.111,E2 -19492.111} C_VEL
LIN {X 0,Y 251.873,Z 358.247,A -85,B 0,C 180,E1 -19493.847,E2 -19493.847} C_VEL
LIN {X 0,Y 257.799,Z 371.218,A -85,B 0,C 180,E1 -19495.401,E2 -19495.401} C_VEL
LIN {X 0,Y 258.724,Z 374.033,A -85,B 0,C 180,E1 -19495.662,E2 -19495.662} C_VEL
LIN {X 0,Y 261.44,Z 391.461,A -85,B 0,C 180,E1 -19496.723,E2 -19496.723} C_VEL
LIN {X 0,Y 259.081,Z 443.047,A -85,B 0,C 180,E1 -19498.129,E2 -19498.129} C_VEL
LIN {X 0,Y 257.65,Z 456.817,A -85,B 0,C 180,E1 -19498.783,E2 -19498.783} C_VEL
LIN {X 0,Y 255.68,Z 469.299,A -85,B 0,C 180,E1 -19499.663,E2 -19499.663} C_VEL
LIN {X 0,Y 253.436,Z 480.433,A -85,B 0,C 180,E1 -19500.741,E2 -19500.741} C_VEL
LIN {X 0,Y 250.666,Z 491.995,A -85,B 0,C 180,E1 -19502.217,E2 -19502.217} C_VEL
LIN {X 0,Y 247.732,Z 502.422,A -85,B 0,C 180,E1 -19503.913,E2 -19503.913} C_VEL
LIN {X 0,Y 244.775,Z 511.84,A -85,B 0,C 180,E1 -19505.848,E2 -19505.848} C_VEL
LIN {X 0,Y 241.629,Z 520.932,A -85,B 0,C 180,E1 -19508.232,E2 -19508.232} C_VEL
LIN {X 0,Y 239.156,Z 528.287,A -85,B 0,C 180,E1 -19510.699,E2 -19510.699} C_VEL
LIN {X 0,Y 236.708,Z 535.061,A -85,B 0,C 180,E1 -19513.616,E2 -19513.616} C_VEL
LIN {X 0,Y 234.984,Z 539.561,A -85,B 0,C 180,E1 -19516.156,E2 -19516.156} C_VEL
LIN {X 0,Y 234.246,Z 541.948,A -85,B 0,C 180,E1 -19517.876,E2 -19517.876} C_VEL
LIN {X 0,Y 233.185,Z 545.47,A -85,B 0,C 180,E1 -19521.332,E2 -19521.332} C_VEL
LIN {X 0,Y 232.732,Z 547.305,A -85,B 0,C 180,E1 -19524.802,E2 -19524.802} C_VEL
LIN {X 0,Y 232.811,Z 547.6,A -85,B 0,C 180,E1 -19528.27,E2 -19528.27} C_VEL
LIN {X 0,Y 232.888,Z 547.133,A -85,B 0,C 180,E1 -19529.999,E2 -19529.999} C_VEL
LIN {X 0,Y 232.836,Z 546.241,A -85,B 0,C 180,E1 -19531.729,E2 -19531.729} C_VEL
LIN {X 0,Y 232.778,Z 543.541,A -85,B 0,C 180,E1 -19534.905,E2 -19534.905} C_VEL
LIN {X 0,Y 233.021,Z 539.789,A -85,B 0,C 180,E1 -19537.8,E2 -19537.8} C_VEL
LIN {X 0,Y 233.468,Z 535.234,A -85,B 0,C 180,E1 -19540.405,E2 -19540.405} C_VEL
LIN {X 0,Y 234.435,Z 528.304,A -85,B 0,C 180,E1 -19543.434,E2 -19543.434} C_VEL
LIN {X 0,Y 235.808,Z 520.783,A -85,B 0,C 180,E1 -19546.002,E2 -19546.002} C_VEL
LIN {X 0,Y 237.413,Z 512.293,A -85,B 0,C 180,E1 -19548.326,E2 -19548.326} C_VEL
LIN {X 0,Y 238.944,Z 502.665,A -85,B 0,C 180,E1 -19550.442,E2 -19550.442} C_VEL
LIN {X 0,Y 240.86,Z 492.034,A -85,B 0,C 180,E1 -19552.291,E2 -19552.291} C_VEL
LIN {X 0,Y 242.762,Z 480.153,A -85,B 0,C 180,E1 -19553.909,E2 -19553.909} C_VEL
LIN {X 0,Y 244.443,Z 467.387,A -85,B 0,C 180,E1 -19555.205,E2 -19555.205} C_VEL
LIN {X 0,Y 245.783,Z 454.621,A -85,B 0,C 180,E1 -19556.137,E2 -19556.137} C_VEL
LIN {X 0,Y 246.617,Z 442.388,A -85,B 0,C 180,E1 -19556.725,E2 -19556.725} C_VEL
LIN {X 0,Y 248.324,Z 386.94,A -85,B 0,C 180,E1 -19558.309,E2 -19558.309} C_VEL
LIN {X 0,Y 244.568,Z 354.753,A -85,B 0,C 180,E1 -19559.728,E2 -19559.728} C_VEL
LIN {X 0,Y 243.673,Z 349.917,A -85,B 0,C 180,E1 -19559.984,E2 -19559.984} C_VEL
LIN {X 0,Y 237.879,Z 334.594,A -85,B 0,C 180,E1 -19561.205,E2 -19561.205} C_VEL
LIN {X 0,Y 235.526,Z 323.603,A -85,B 0,C 180,E1 -19565.564,E2 -19565.564} C_VEL
LIN {X 0,Y 234.998,Z 321.213,A -85,B 0,C 180,E1 -19566.552,E2 -19566.552} C_VEL
LIN {X 0,Y 234.88,Z 321.227,A -85,B 0,C 180,E1 -19571.167,E2 -19571.167} C_VEL
LIN {X 0,Y 234.883,Z 321.227,A -85,B 0,C 180,E1 -19575.897,E2 -19575.897} C_VEL
LIN {X 0,Y 234.88,Z 321.229,A -85,B 0,C 180,E1 -19578.831,E2 -19578.831} C_VEL
LIN {X 0,Y 234.916,Z 321.225,A -85,B 0,C 180,E1 -19581.078,E2 -19581.078} C_VEL
LIN {X 0,Y 234.925,Z 321.223,A -85,B 0,C 180,E1 -19585.361,E2 -19585.361} C_VEL
LIN {X 0,Y 234.929,Z 321.223,A -85,B 0,C 180,E1 -19589.431,E2 -19589.431} C_VEL
LIN {X 0,Y 234.992,Z 321.213,A -85,B 0,C 180,E1 -19593.793,E2 -19593.793} C_VEL
LIN {X 0,Y 235.009,Z 321.211,A -85,B 0,C 180,E1 -19598.969,E2 -19598.969} C_VEL
LIN {X 0,Y 235.093,Z 321.2,A -85,B 0,C 180,E1 -19603.059,E2 -19603.059} C_VEL
LIN {X 0,Y 235.115,Z 321.182,A -85,B 0,C 180,E1 -19607.922,E2 -19607.922} C_VEL
LIN {X 0,Y 235.372,Z 321.16,A -85,B 0,C 180,E1 -19611.414,E2 -19611.414} C_VEL
LIN {X 0,Y 235.399,Z 321.161,A -85,B 0,C 180,E1 -19613.141,E2 -19613.141} C_VEL
LIN {X 0,Y 235.592,Z 321.122,A -85,B 0,C 180,E1 -19618.29,E2 -19618.29} C_VEL
LIN {X 0,Y 235.591,Z 321.131,A -85,B 0,C 180,E1 -19621.709,E2 -19621.709} C_VEL
LIN {X 0,Y 235.355,Z 321.162,A -85,B 0,C 180,E1 -19626.86,E2 -19626.86} C_VEL
LIN {X 0,Y 235.21,Z 321.17,A -85,B 0,C 180,E1 -19630.327,E2 -19630.327} C_VEL
LIN {X 0,Y 235.11,Z 321.198,A -85,B 0,C 180,E1 -19635.606,E2 -19635.606} C_VEL
LIN {X 0,Y 235.003,Z 321.198,A -85,B 0,C 180,E1 -19639.206,E2 -19639.206} C_VEL
LIN {X 0,Y 234.949,Z 321.215,A -85,B 0,C 180,E1 -19642.884,E2 -19642.884} C_VEL
LIN {X 0,Y 234.966,Z 321.214,A -85,B 0,C 180,E1 -19646.657,E2 -19646.657} C_VEL
LIN {X 0,Y 234.928,Z 321.206,A -85,B 0,C 180,E1 -19650.568,E2 -19650.568} C_VEL
LIN {X 0,Y 234.926,Z 321.222,A -85,B 0,C 180,E1 -19654.638,E2 -19654.638} C_VEL
LIN {X 0,Y 234.938,Z 321.207,A -85,B 0,C 180,E1 -19658.945,E2 -19658.945} C_VEL
LIN {X 0,Y 234.872,Z 321.224,A -85,B 0,C 180,E1 -19663.489,E2 -19663.489} C_VEL
LIN {X 0,Y 234.854,Z 321.219,A -85,B 0,C 180,E1 -19666.508,E2 -19666.508} C_VEL
LIN {X 0,Y 234.914,Z 321.218,A -85,B 0,C 180,E1 -19671.079,E2 -19671.079} C_VEL
LIN {X 0,Y 234.926,Z 321.222,A -85,B 0,C 180,E1 -19675.362,E2 -19675.362} C_VEL
LIN {X 0,Y 234.892,Z 321.221,A -85,B 0,C 180,E1 -19679.428,E2 -19679.428} C_VEL
LIN {X 0,Y 234.938,Z 321.218,A -85,B 0,C 180,E1 -19683.822,E2 -19683.822} C_VEL
LIN {X 0,Y 234.989,Z 321.214,A -85,B 0,C 180,E1 -19688.58,E2 -19688.58} C_VEL
LIN {X 0,Y 236.123,Z 324.263,A -85,B 0,C 180,E1 -19688.864,E2 -19688.864} C_VEL
LIN {X 0,Y 241.919,Z 336.28,A -85,B 0,C 180,E1 -19689.964,E2 -19689.964} C_VEL
LIN {X 0,Y 248.422,Z 353.527,A -85,B 0,C 180,E1 -19691.246,E2 -19691.246} C_VEL
LIN {X 0,Y 249.262,Z 356.427,A -85,B 0,C 180,E1 -19691.427,E2 -19691.427} C_VEL
LIN {X 0,Y 246.97,Z 426.817,A -85,B 0,C 180,E1 -19693.433,E2 -19693.433} C_VEL
LIN {X 0,Y 246.146,Z 440.37,A -85,B 0,C 180,E1 -19694.156,E2 -19694.156} C_VEL
LIN {X 0,Y 245.029,Z 452.845,A -85,B 0,C 180,E1 -19695.147,E2 -19695.147} C_VEL
LIN {X 0,Y 243.609,Z 464.767,A -85,B 0,C 180,E1 -19696.444,E2 -19696.444} C_VEL
LIN {X 0,Y 241.744,Z 474.968,A -85,B 0,C 180,E1 -19697.833,E2 -19697.833} C_VEL
LIN {X 0,Y 240.044,Z 485.462,A -85,B 0,C 180,E1 -19699.67,E2 -19699.67} C_VEL
LIN {X 0,Y 238.431,Z 494.062,A -85,B 0,C 180,E1 -19701.526,E2 -19701.526} C_VEL
LIN {X 0,Y 237.008,Z 501.97,A -85,B 0,C 180,E1 -19703.616,E2 -19703.616} C_VEL
LIN {X 0,Y 235.485,Z 509.733,A -85,B 0,C 180,E1 -19706.15,E2 -19706.15} C_VEL
LIN {X 0,Y 234.259,Z 516.841,A -85,B 0,C 180,E1 -19709.141,E2 -19709.141} C_VEL
LIN {X 0,Y 233.47,Z 521.596,A -85,B 0,C 180,E1 -19711.726,E2 -19711.726} C_VEL
LIN {X 0,Y 233.177,Z 525.231,A -85,B 0,C 180,E1 -19714.322,E2 -19714.322} C_VEL
LIN {X 0,Y 232.867,Z 527.875,A -85,B 0,C 180,E1 -19716.934,E2 -19716.934} C_VEL
LIN {X 0,Y 232.673,Z 529.133,A -85,B 0,C 180,E1 -19718.687,E2 -19718.687} C_VEL
LIN {X 0,Y 232.641,Z 529.962,A -85,B 0,C 180,E1 -19720.444,E2 -19720.444} C_VEL
LIN {X 0,Y 232.952,Z 530.385,A -85,B 0,C 180,E1 -19723.967,E2 -19723.967} C_VEL
LIN {X 0,Y 233.297,Z 530.012,A -85,B 0,C 180,E1 -19725.732,E2 -19725.732} C_VEL
LIN {X 0,Y 233.681,Z 529.205,A -85,B 0,C 180,E1 -19727.503,E2 -19727.503} C_VEL
LIN {X 0,Y 234.248,Z 527.968,A -85,B 0,C 180,E1 -19729.271,E2 -19729.271} C_VEL
LIN {X 0,Y 235.7,Z 524.675,A -85,B 0,C 180,E1 -19732.431,E2 -19732.431} C_VEL
LIN {X 0,Y 237.631,Z 520.121,A -85,B 0,C 180,E1 -19735.395,E2 -19735.395} C_VEL
LIN {X 0,Y 239.683,Z 514.795,A -85,B 0,C 180,E1 -19737.98,E2 -19737.98} C_VEL
LIN {X 0,Y 242.228,Z 508.063,A -85,B 0,C 180,E1 -19740.514,E2 -19740.514} C_VEL
LIN {X 0,Y 245.194,Z 499.653,A -85,B 0,C 180,E1 -19742.998,E2 -19742.998} C_VEL
LIN {X 0,Y 248.035,Z 490.943,A -85,B 0,C 180,E1 -19745.014,E2 -19745.014} C_VEL
LIN {X 0,Y 251.086,Z 480.12,A -85,B 0,C 180,E1 -19746.999,E2 -19746.999} C_VEL
LIN {X 0,Y 253.669,Z 469.299,A -85,B 0,C 180,E1 -19748.563,E2 -19748.563} C_VEL
LIN {X 0,Y 256.009,Z 457.264,A -85,B 0,C 180,E1 -19749.897,E2 -19749.897} C_VEL
LIN {X 0,Y 257.76,Z 445.585,A -85,B 0,C 180,E1 -19750.873,E2 -19750.873} C_VEL
LIN {X 0,Y 259.014,Z 433.206,A -85,B 0,C 180,E1 -19751.623,E2 -19751.623} C_VEL
LIN {X 0,Y 259.985,Z 420.889,A -85,B 0,C 180,E1 -19752.056,E2 -19752.056} C_VEL
LIN {X 0,Y 262.308,Z 370.35,A -85,B 0,C 180,E1 -19753.385,E2 -19753.385} C_VEL
LIN {X 0,Y 255.32,Z 355.429,A -85,B 0,C 180,E1 -19755.142,E2 -19755.142} C_VEL
LIN {X 0,Y 248.824,Z 343.462,A -85,B 0,C 180,E1 -19756.839,E2 -19756.839} C_VEL
LIN {X 0,Y 244.826,Z 336.811,A -85,B 0,C 180,E1 -19757.925,E2 -19757.925} C_VEL
LIN {X 0,Y 240.173,Z 329.858,A -85,B 0,C 180,E1 -19759.231,E2 -19759.231} C_VEL
LIN {X 0,Y 238.02,Z 326.47,A -85,B 0,C 180,E1 -19759.871,E2 -19759.871} C_VEL
LIN {X 0,Y 235.626,Z 323.56,A -85,B 0,C 180,E1 -19760.568,E2 -19760.568} C_VEL
LIN {X 0,Y 234.938,Z 321.217,A -85,B 0,C 180,E1 -19760.86,E2 -19760.86} C_VEL
LIN {X 0,Y 234.931,Z 321.214,A -85,B 0,C 180,E1 -19765.362,E2 -19765.362} C_VEL
LIN {X 0,Y 234.932,Z 321.205,A -85,B 0,C 180,E1 -19769.433,E2 -19769.433} C_VEL
LIN {X 0,Y 234.995,Z 321.202,A -85,B 0,C 180,E1 -19773.794,E2 -19773.794} C_VEL
LIN {X 0,Y 234.998,Z 321.209,A -85,B 0,C 180,E1 -19778.969,E2 -19778.969} C_VEL
LIN {X 0,Y 235.097,Z 321.201,A -85,B 0,C 180,E1 -19783.06,E2 -19783.06} C_VEL
LIN {X 0,Y 235.148,Z 321.189,A -85,B 0,C 180,E1 -19787.924,E2 -19787.924} C_VEL
LIN {X 0,Y 235.391,Z 321.164,A -85,B 0,C 180,E1 -19791.415,E2 -19791.415} C_VEL
LIN {X 0,Y 235.406,Z 321.151,A -85,B 0,C 180,E1 -19793.142,E2 -19793.142} C_VEL
LIN {X 0,Y 235.596,Z 321.126,A -85,B 0,C 180,E1 -19798.291,E2 -19798.291} C_VEL
LIN {X 0,Y 235.596,Z 321.128,A -85,B 0,C 180,E1 -19801.71,E2 -19801.71} C_VEL
LIN {X 0,Y 235.405,Z 321.147,A -85,B 0,C 180,E1 -19806.859,E2 -19806.859} C_VEL
LIN {X 0,Y 235.24,Z 321.175,A -85,B 0,C 180,E1 -19810.327,E2 -19810.327} C_VEL
LIN {X 0,Y 235.116,Z 321.186,A -85,B 0,C 180,E1 -19815.607,E2 -19815.607} C_VEL
LIN {X 0,Y 235.09,Z 321.188,A -85,B 0,C 180,E1 -19816.345,E2 -19816.345} C_VEL
LIN {X 0,Y 234.415,Z 321.282,A -85,B 0,C 180,E1 -19817.774,E2 -19817.774} C_VEL
LIN {X 0,Y 231.531,Z 321.643,A -85,B 0,C 180,E1 -19820.103,E2 -19820.103} C_VEL
LIN {X 0,Y 229.067,Z 321.95,A -85,B 0,C 180,E1 -19822.001,E2 -19822.001} C_VEL
LIN {X 0,Y 227.99,Z 322.081,A -85,B 0,C 180,E1 -19823.476,E2 -19823.476} C_VEL
LIN {X 0,Y 227.893,Z 322.089,A -85,B 0,C 180,E1 -19823.977,E2 -19823.977} C_VEL
LIN {X 0,Y 227.881,Z 322.095,A -85,B 0,C 180,E1 -19827.556,E2 -19827.556} C_VEL
LIN {X 0,Y 227.869,Z 322.094,A -85,B 0,C 180,E1 -19831.623,E2 -19831.623} C_VEL
LIN {X 0,Y 227.882,Z 322.09,A -85,B 0,C 180,E1 -19835.872,E2 -19835.872} C_VEL
LIN {X 0,Y 227.813,Z 322.077,A -85,B 0,C 180,E1 -19840.38,E2 -19840.38} C_VEL
LIN {X 0,Y 227.812,Z 322.128,A -85,B 0,C 180,E1 -19842.089,E2 -19842.089} C_VEL
LIN {X 0,Y 230.122,Z 329.673,A -85,B 0,C 180,E1 -19846.497,E2 -19846.497} C_VEL
LIN {X 0,Y 231.114,Z 333.007,A -85,B 0,C 180,E1 -19848.25,E2 -19848.25} C_VEL
LIN {X 0,Y 233.468,Z 337.184,A -85,B 0,C 180,E1 -19849.022,E2 -19849.022} C_VEL
LIN {X 0,Y 234.887,Z 339.539,A -85,B 0,C 180,E1 -19849.467,E2 -19849.467} C_VEL
LIN {X 0,Y 238.267,Z 345.316,A -85,B 0,C 180,E1 -19850.501,E2 -19850.501} C_VEL
LIN {X 0,Y 244.57,Z 357.095,A -85,B 0,C 180,E1 -19852.346,E2 -19852.346} C_VEL
LIN {X 0,Y 251.133,Z 370.982,A -85,B 0,C 180,E1 -19854.173,E2 -19854.173} C_VEL
LIN {X 0,Y 253.355,Z 376.628,A -85,B 0,C 180,E1 -19854.793,E2 -19854.793} C_VEL
LIN {X 0,Y 255.708,Z 392.306,A -85,B 0,C 180,E1 -19855.773,E2 -19855.773} C_VEL
LIN {X 0,Y 253.382,Z 442.655,A -85,B 0,C 180,E1 -19857.18,E2 -19857.18} C_VEL
LIN {X 0,Y 251.972,Z 456.036,A -85,B 0,C 180,E1 -19857.82,E2 -19857.82} C_VEL
LIN {X 0,Y 249.821,Z 469.213,A -85,B 0,C 180,E1 -19858.755,E2 -19858.755} C_VEL
LIN {X 0,Y 247.303,Z 481.085,A -85,B 0,C 180,E1 -19859.942,E2 -19859.942} C_VEL
LIN {X 0,Y 244.429,Z 492.48,A -85,B 0,C 180,E1 -19861.444,E2 -19861.444} C_VEL
LIN {X 0,Y 241.394,Z 502.776,A -85,B 0,C 180,E1 -19863.174,E2 -19863.174} C_VEL
LIN {X 0,Y 238.318,Z 512.049,A -85,B 0,C 180,E1 -19865.15,E2 -19865.15} C_VEL
LIN {X 0,Y 235.045,Z 521.054,A -85,B 0,C 180,E1 -19867.59,E2 -19867.59} C_VEL
LIN {X 0,Y 232.47,Z 528.327,A -85,B 0,C 180,E1 -19870.116,E2 -19870.116} C_VEL
LIN {X 0,Y 229.893,Z 535.023,A -85,B 0,C 180,E1 -19873.116,E2 -19873.116} C_VEL
LIN {X 0,Y 228.066,Z 539.471,A -85,B 0,C 180,E1 -19875.728,E2 -19875.728} C_VEL
LIN {X 0,Y 227.274,Z 541.833,A -85,B 0,C 180,E1 -19877.498,E2 -19877.498} C_VEL
LIN {X 0,Y 226.609,Z 543.773,A -85,B 0,C 180,E1 -19879.275,E2 -19879.275} C_VEL
LIN {X 0,Y 226.143,Z 545.295,A -85,B 0,C 180,E1 -19881.06,E2 -19881.06} C_VEL
LIN {X 0,Y 225.648,Z 547.073,A -85,B 0,C 180,E1 -19884.638,E2 -19884.638} C_VEL
LIN {X 0,Y 225.626,Z 547.389,A -85,B 0,C 180,E1 -19886.428,E2 -19886.428} C_VEL
LIN {X 0,Y 225.72,Z 547.319,A -85,B 0,C 180,E1 -19888.215,E2 -19888.215} C_VEL
LIN {X 0,Y 225.819,Z 546.813,A -85,B 0,C 180,E1 -19889.999,E2 -19889.999} C_VEL
LIN {X 0,Y 225.747,Z 545.897,A -85,B 0,C 180,E1 -19891.783,E2 -19891.783} C_VEL
LIN {X 0,Y 225.69,Z 543.408,A -85,B 0,C 180,E1 -19894.802,E2 -19894.802} C_VEL
LIN {X 0,Y 225.958,Z 539.342,A -85,B 0,C 180,E1 -19898.045,E2 -19898.045} C_VEL
LIN {X 0,Y 226.441,Z 534.728,A -85,B 0,C 180,E1 -19900.732,E2 -19900.732} C_VEL
LIN {X 0,Y 227.498,Z 527.72,A -85,B 0,C 180,E1 -19903.851,E2 -19903.851} C_VEL
LIN {X 0,Y 228.916,Z 520.128,A -85,B 0,C 180,E1 -19906.497,E2 -19906.497} C_VEL
LIN {X 0,Y 230.347,Z 513.089,A -85,B 0,C 180,E1 -19908.484,E2 -19908.484} C_VEL
LIN {X 0,Y 232.047,Z 502.868,A -85,B 0,C 180,E1 -19910.846,E2 -19910.846} C_VEL
LIN {X 0,Y 234.033,Z 492.335,A -85,B 0,C 180,E1 -19912.744,E2 -19912.744} C_VEL
LIN {X 0,Y 235.991,Z 480.613,A -85,B 0,C 180,E1 -19914.406,E2 -19914.406} C_VEL
LIN {X 0,Y 237.721,Z 468.109,A -85,B 0,C 180,E1 -19915.735,E2 -19915.735} C_VEL
LIN {X 0,Y 239.178,Z 454.919,A -85,B 0,C 180,E1 -19916.739,E2 -19916.739} C_VEL
LIN {X 0,Y 240.089,Z 441.706,A -85,B 0,C 180,E1 -19917.394,E2 -19917.394} C_VEL
LIN {X 0,Y 241.828,Z 387.017,A -85,B 0,C 180,E1 -19918.994,E2 -19918.994} C_VEL
LIN {X 0,Y 237.876,Z 353.422,A -85,B 0,C 180,E1 -19920.539,E2 -19920.539} C_VEL
LIN {X 0,Y 232.024,Z 337.968,A -85,B 0,C 180,E1 -19921.78,E2 -19921.78} C_VEL
LIN {X 0,Y 230.59,Z 334.304,A -85,B 0,C 180,E1 -19922.131,E2 -19922.131} C_VEL
LIN {X 0,Y 228.726,Z 325.581,A -85,B 0,C 180,E1 -19925.718,E2 -19925.718} C_VEL
LIN {X 0,Y 227.895,Z 322.097,A -85,B 0,C 180,E1 -19927.23,E2 -19927.23} C_VEL
LIN {X 0,Y 227.824,Z 322.108,A -85,B 0,C 180,E1 -19930.376,E2 -19930.376} C_VEL
LIN {X 0,Y 227.824,Z 322.106,A -85,B 0,C 180,E1 -19935.194,E2 -19935.194} C_VEL
LIN {X 0,Y 227.823,Z 322.106,A -85,B 0,C 180,E1 -19939.622,E2 -19939.622} C_VEL
LIN {X 0,Y 227.878,Z 322.102,A -85,B 0,C 180,E1 -19944.127,E2 -19944.127} C_VEL
LIN {X 0,Y 227.868,Z 322.101,A -85,B 0,C 180,E1 -19948.377,E2 -19948.377} C_VEL
LIN {X 0,Y 227.884,Z 322.099,A -85,B 0,C 180,E1 -19952.444,E2 -19952.444} C_VEL
LIN {X 0,Y 227.912,Z 322.095,A -85,B 0,C 180,E1 -19956.367,E2 -19956.367} C_VEL
LIN {X 0,Y 227.94,Z 322.09,A -85,B 0,C 180,E1 -19960.174,E2 -19960.174} C_VEL
LIN {X 0,Y 228.055,Z 322.076,A -85,B 0,C 180,E1 -19963.897,E2 -19963.897} C_VEL
LIN {X 0,Y 228.072,Z 322.061,A -85,B 0,C 180,E1 -19967.543,E2 -19967.543} C_VEL
LIN {X 0,Y 228.302,Z 322.038,A -85,B 0,C 180,E1 -19971.145,E2 -19971.145} C_VEL
LIN {X 0,Y 228.35,Z 322.038,A -85,B 0,C 180,E1 -19972.928,E2 -19972.928} C_VEL
LIN {X 0,Y 228.55,Z 321.999,A -85,B 0,C 180,E1 -19978.237,E2 -19978.237} C_VEL
LIN {X 0,Y 228.549,Z 322.008,A -85,B 0,C 180,E1 -19981.762,E2 -19981.762} C_VEL
LIN {X 0,Y 228.307,Z 322.04,A -85,B 0,C 180,E1 -19987.073,E2 -19987.073} C_VEL
LIN {X 0,Y 228.142,Z 322.051,A -85,B 0,C 180,E1 -19990.651,E2 -19990.651} C_VEL
LIN {X 0,Y 228.061,Z 322.078,A -85,B 0,C 180,E1 -19994.272,E2 -19994.272} C_VEL
LIN {X 0,Y 227.999,Z 322.078,A -85,B 0,C 180,E1 -19997.953,E2 -19997.953} C_VEL
LIN {X 0,Y 227.913,Z 322.085,A -85,B 0,C 180,E1 -20002.321,E2 -20002.321} C_VEL
LIN {X 0,Y 227.939,Z 322.09,A -85,B 0,C 180,E1 -20006.603,E2 -20006.603} C_VEL
LIN {X 0,Y 227.905,Z 322.079,A -85,B 0,C 180,E1 -20010.296,E2 -20010.296} C_VEL
LIN {X 0,Y 227.873,Z 322.096,A -85,B 0,C 180,E1 -20013.721,E2 -20013.721} C_VEL
LIN {X 0,Y 227.84,Z 322.092,A -85,B 0,C 180,E1 -20018.091,E2 -20018.091} C_VEL
LIN {X 0,Y 227.801,Z 322.109,A -85,B 0,C 180,E1 -20022.744,E2 -20022.744} C_VEL
LIN {X 0,Y 227.784,Z 322.105,A -85,B 0,C 180,E1 -20027.253,E2 -20027.253} C_VEL
LIN {X 0,Y 227.84,Z 322.097,A -85,B 0,C 180,E1 -20031.909,E2 -20031.909} C_VEL
LIN {X 0,Y 227.876,Z 322.098,A -85,B 0,C 180,E1 -20036.378,E2 -20036.378} C_VEL
LIN {X 0,Y 227.869,Z 322.094,A -85,B 0,C 180,E1 -20040.432,E2 -20040.432} C_VEL
LIN {X 0,Y 227.872,Z 322.097,A -85,B 0,C 180,E1 -20044.42,E2 -20044.42} C_VEL
LIN {X 0,Y 227.936,Z 322.093,A -85,B 0,C 180,E1 -20047.718,E2 -20047.718} C_VEL
LIN {X 0,Y 228.991,Z 325.036,A -85,B 0,C 180,E1 -20047.967,E2 -20047.967} C_VEL
LIN {X 0,Y 235.766,Z 338.681,A -85,B 0,C 180,E1 -20049.306,E2 -20049.306} C_VEL
LIN {X 0,Y 242.512,Z 356.664,A -85,B 0,C 180,E1 -20050.693,E2 -20050.693} C_VEL
LIN {X 0,Y 242.724,Z 360.032,A -85,B 0,C 180,E1 -20050.826,E2 -20050.826} C_VEL
LIN {X 0,Y 240.418,Z 427.524,A -85,B 0,C 180,E1 -20052.804,E2 -20052.804} C_VEL
LIN {X 0,Y 239.572,Z 440.926,A -85,B 0,C 180,E1 -20053.545,E2 -20053.545} C_VEL
LIN {X 0,Y 238.359,Z 453.836,A -85,B 0,C 180,E1 -20054.612,E2 -20054.612} C_VEL
LIN {X 0,Y 236.726,Z 466.371,A -85,B 0,C 180,E1 -20056.042,E2 -20056.042} C_VEL
LIN {X 0,Y 234.807,Z 476.328,A -85,B 0,C 180,E1 -20057.468,E2 -20057.468} C_VEL
LIN {X 0,Y 233.114,Z 486.625,A -85,B 0,C 180,E1 -20059.359,E2 -20059.359} C_VEL
LIN {X 0,Y 231.437,Z 495.078,A -85,B 0,C 180,E1 -20061.267,E2 -20061.267} C_VEL
LIN {X 0,Y 229.708,Z 504.214,A -85,B 0,C 180,E1 -20063.853,E2 -20063.853} C_VEL
LIN {X 0,Y 228.179,Z 511.585,A -85,B 0,C 180,E1 -20066.469,E2 -20066.469} C_VEL
LIN {X 0,Y 227.164,Z 517.488,A -85,B 0,C 180,E1 -20069.114,E2 -20069.114} C_VEL
LIN {X 0,Y 226.368,Z 522.163,A -85,B 0,C 180,E1 -20071.78,E2 -20071.78} C_VEL
LIN {X 0,Y 226.06,Z 525.723,A -85,B 0,C 180,E1 -20074.458,E2 -20074.458} C_VEL
LIN {X 0,Y 225.753,Z 528.297,A -85,B 0,C 180,E1 -20077.154,E2 -20077.154} C_VEL
LIN {X 0,Y 225.578,Z 529.514,A -85,B 0,C 180,E1 -20078.962,E2 -20078.962} C_VEL
LIN {X 0,Y 225.547,Z 530.281,A -85,B 0,C 180,E1 -20080.776,E2 -20080.776} C_VEL
LIN {X 0,Y 225.946,Z 530.636,A -85,B 0,C 180,E1 -20084.409,E2 -20084.409} C_VEL
LIN {X 0,Y 226.301,Z 530.218,A -85,B 0,C 180,E1 -20086.231,E2 -20086.231} C_VEL
LIN {X 0,Y 226.73,Z 529.353,A -85,B 0,C 180,E1 -20088.058,E2 -20088.058} C_VEL
LIN {X 0,Y 227.369,Z 528.081,A -85,B 0,C 180,E1 -20089.878,E2 -20089.878} C_VEL
LIN {X 0,Y 228.818,Z 525.027,A -85,B 0,C 180,E1 -20092.865,E2 -20092.865} C_VEL
LIN {X 0,Y 230.373,Z 521.554,A -85,B 0,C 180,E1 -20095.284,E2 -20095.284} C_VEL
LIN {X 0,Y 232.479,Z 516.581,A -85,B 0,C 180,E1 -20097.942,E2 -20097.942} C_VEL
LIN {X 0,Y 235.029,Z 510.274,A -85,B 0,C 180,E1 -20100.554,E2 -20100.554} C_VEL
LIN {X 0,Y 238.009,Z 502.314,A -85,B 0,C 180,E1 -20103.112,E2 -20103.112} C_VEL
LIN {X 0,Y 240.962,Z 493.864,A -85,B 0,C 180,E1 -20105.249,E2 -20105.249} C_VEL
LIN {X 0,Y 244.035,Z 484.102,A -85,B 0,C 180,E1 -20107.214,E2 -20107.214} C_VEL
LIN {X 0,Y 246.609,Z 474.162,A -85,B 0,C 180,E1 -20108.827,E2 -20108.827} C_VEL
LIN {X 0,Y 249.213,Z 462.742,A -85,B 0,C 180,E1 -20110.255,E2 -20110.255} C_VEL
LIN {X 0,Y 251.243,Z 450.662,A -85,B 0,C 180,E1 -20111.433,E2 -20111.433} C_VEL
LIN {X 0,Y 252.886,Z 437.815,A -85,B 0,C 180,E1 -20112.331,E2 -20112.331} C_VEL
LIN {X 0,Y 253.975,Z 425.342,A -85,B 0,C 180,E1 -20112.881,E2 -20112.881} C_VEL
LIN {X 0,Y 256.578,Z 372.436,A -85,B 0,C 180,E1 -20114.308,E2 -20114.308} C_VEL
LIN {X 0,Y 249.845,Z 358.093,A -85,B 0,C 180,E1 -20116.087,E2 -20116.087} C_VEL
LIN {X 0,Y 241.758,Z 343.251,A -85,B 0,C 180,E1 -20118.335,E2 -20118.335} C_VEL
LIN {X 0,Y 235.907,Z 334.622,A -85,B 0,C 180,E1 -20120.031,E2 -20120.031} C_VEL
LIN {X 0,Y 233.336,Z 330.903,A -85,B 0,C 180,E1 -20120.817,E2 -20120.817} C_VEL
LIN {X 0,Y 231.158,Z 327.508,A -85,B 0,C 180,E1 -20121.516,E2 -20121.516} C_VEL
LIN {X 0,Y 228.728,Z 324.757,A -85,B 0,C 180,E1 -20122.276,E2 -20122.276} C_VEL
LIN {X 0,Y 227.866,Z 322.096,A -85,B 0,C 180,E1 -20122.687,E2 -20122.687} C_VEL
LIN {X 0,Y 227.88,Z 322.091,A -85,B 0,C 180,E1 -20126.378,E2 -20126.378} C_VEL
LIN {X 0,Y 227.92,Z 322.085,A -85,B 0,C 180,E1 -20130.438,E2 -20130.438} C_VEL
LIN {X 0,Y 227.926,Z 322.087,A -85,B 0,C 180,E1 -20134.426,E2 -20134.426} C_VEL
LIN {X 0,Y 227.948,Z 322.087,A -85,B 0,C 180,E1 -20138.286,E2 -20138.286} C_VEL
LIN {X 0,Y 228.035,Z 322.08,A -85,B 0,C 180,E1 -20142.826,E2 -20142.826} C_VEL
LIN {X 0,Y 228.095,Z 322.07,A -85,B 0,C 180,E1 -20147.545,E2 -20147.545} C_VEL
LIN {X 0,Y 228.326,Z 322.043,A -85,B 0,C 180,E1 -20151.147,E2 -20151.147} C_VEL
LIN {X 0,Y 228.359,Z 322.03,A -85,B 0,C 180,E1 -20152.929,E2 -20152.929} C_VEL
LIN {X 0,Y 228.555,Z 322.002,A -85,B 0,C 180,E1 -20158.238,E2 -20158.238} C_VEL
LIN {X 0,Y 228.555,Z 322.004,A -85,B 0,C 180,E1 -20161.762,E2 -20161.762} C_VEL
LIN {X 0,Y 228.356,Z 322.024,A -85,B 0,C 180,E1 -20167.072,E2 -20167.072} C_VEL
LIN {X 0,Y 228.161,Z 322.054,A -85,B 0,C 180,E1 -20170.651,E2 -20170.651} C_VEL
LIN {X 0,Y 228.067,Z 322.074,A -85,B 0,C 180,E1 -20174.272,E2 -20174.272} C_VEL
LIN {X 0,Y 228.005,Z 322.081,A -85,B 0,C 180,E1 -20177.954,E2 -20177.954} C_VEL
LIN {X 0,Y 227.919,Z 322.093,A -85,B 0,C 180,E1 -20182.321,E2 -20182.321} C_VEL
LIN {X 0,Y 227.893,Z 322.089,A -85,B 0,C 180,E1 -20183.977,E2 -20183.977} C_VEL
LIN {X 0,Y 227.195,Z 322.18,A -85,B 0,C 180,E1 -20185.451,E2 -20185.451} C_VEL
LIN {X 0,Y 224.328,Z 322.535,A -85,B 0,C 180,E1 -20187.857,E2 -20187.857} C_VEL
LIN {X 0,Y 221.911,Z 322.839,A -85,B 0,C 180,E1 -20189.82,E2 -20189.82} C_VEL
LIN {X 0,Y 220.878,Z 322.968,A -85,B 0,C 180,E1 -20191.344,E2 -20191.344} C_VEL
LIN {X 0,Y 220.795,Z 322.973,A -85,B 0,C 180,E1 -20191.861,E2 -20191.861} C_VEL
LIN {X 0,Y 220.803,Z 322.975,A -85,B 0,C 180,E1 -20194.955,E2 -20194.955} C_VEL
LIN {X 0,Y 220.812,Z 322.977,A -85,B 0,C 180,E1 -20197.278,E2 -20197.278} C_VEL
LIN {X 0,Y 220.813,Z 323.151,A -85,B 0,C 180,E1 -20200.497,E2 -20200.497} C_VEL
LIN {X 0,Y 223.087,Z 330.608,A -85,B 0,C 180,E1 -20205.14,E2 -20205.14} C_VEL
LIN {X 0,Y 223.75,Z 332.643,A -85,B 0,C 180,E1 -20206.256,E2 -20206.256} C_VEL
LIN {X 0,Y 226.491,Z 337.237,A -85,B 0,C 180,E1 -20207.227,E2 -20207.227} C_VEL
LIN {X 0,Y 227.954,Z 339.667,A -85,B 0,C 180,E1 -20207.727,E2 -20207.727} C_VEL
LIN {X 0,Y 231.059,Z 344.845,A -85,B 0,C 180,E1 -20208.755,E2 -20208.755} C_VEL
LIN {X 0,Y 235.676,Z 352.841,A -85,B 0,C 180,E1 -20210.213,E2 -20210.213} C_VEL
LIN {X 0,Y 243.673,Z 368.945,A -85,B 0,C 180,E1 -20212.618,E2 -20212.618} C_VEL
LIN {X 0,Y 248.013,Z 379.096,A -85,B 0,C 180,E1 -20213.874,E2 -20213.874} C_VEL
LIN {X 0,Y 250.127,Z 393.268,A -85,B 0,C 180,E1 -20214.798,E2 -20214.798} C_VEL
LIN {X 0,Y 247.788,Z 442.025,A -85,B 0,C 180,E1 -20216.18,E2 -20216.18} C_VEL
LIN {X 0,Y 246.312,Z 455.587,A -85,B 0,C 180,E1 -20216.831,E2 -20216.831} C_VEL
LIN {X 0,Y 244.231,Z 468.021,A -85,B 0,C 180,E1 -20217.713,E2 -20217.713} C_VEL
LIN {X 0,Y 241.621,Z 480.162,A -85,B 0,C 180,E1 -20218.916,E2 -20218.916} C_VEL
LIN {X 0,Y 238.596,Z 491.68,A -85,B 0,C 180,E1 -20220.436,E2 -20220.436} C_VEL
LIN {X 0,Y 235.423,Z 502.067,A -85,B 0,C 180,E1 -20222.196,E2 -20222.196} C_VEL
LIN {X 0,Y 232.525,Z 510.575,A -85,B 0,C 180,E1 -20224.007,E2 -20224.007} C_VEL
LIN {X 0,Y 229.571,Z 518.441,A -85,B 0,C 180,E1 -20226.069,E2 -20226.069} C_VEL
LIN {X 0,Y 226.543,Z 526.395,A -85,B 0,C 180,E1 -20228.725,E2 -20228.725} C_VEL
LIN {X 0,Y 223.801,Z 533.272,A -85,B 0,C 180,E1 -20231.697,E2 -20231.697} C_VEL
LIN {X 0,Y 221.77,Z 538.042,A -85,B 0,C 180,E1 -20234.373,E2 -20234.373} C_VEL
LIN {X 0,Y 220.296,Z 541.719,A -85,B 0,C 180,E1 -20237.095,E2 -20237.095} C_VEL
LIN {X 0,Y 219.619,Z 543.635,A -85,B 0,C 180,E1 -20238.93,E2 -20238.93} C_VEL
LIN {X 0,Y 219.095,Z 545.11,A -85,B 0,C 180,E1 -20240.77,E2 -20240.77} C_VEL
LIN {X 0,Y 218.571,Z 546.842,A -85,B 0,C 180,E1 -20244.464,E2 -20244.464} C_VEL
LIN {X 0,Y 218.525,Z 547.135,A -85,B 0,C 180,E1 -20246.311,E2 -20246.311} C_VEL
LIN {X 0,Y 218.632,Z 547.028,A -85,B 0,C 180,E1 -20248.157,E2 -20248.157} C_VEL
LIN {X 0,Y 218.751,Z 546.493,A -85,B 0,C 180,E1 -20249.999,E2 -20249.999} C_VEL
LIN {X 0,Y 218.66,Z 545.553,A -85,B 0,C 180,E1 -20251.841,E2 -20251.841} C_VEL
LIN {X 0,Y 218.59,Z 543.315,A -85,B 0,C 180,E1 -20254.652,E2 -20254.652} C_VEL
LIN {X 0,Y 218.792,Z 540.162,A -85,B 0,C 180,E1 -20257.381,E2 -20257.381} C_VEL
LIN {X 0,Y 219.212,Z 535.877,A -85,B 0,C 180,E1 -20260.155,E2 -20260.155} C_VEL
LIN {X 0,Y 220.167,Z 529.365,A -85,B 0,C 180,E1 -20263.38,E2 -20263.38} C_VEL
LIN {X 0,Y 221.58,Z 522.223,A -85,B 0,C 180,E1 -20266.112,E2 -20266.112} C_VEL
LIN {X 0,Y 223.283,Z 513.842,A -85,B 0,C 180,E1 -20268.662,E2 -20268.662} C_VEL
LIN {X 0,Y 225.032,Z 504.095,A -85,B 0,C 180,E1 -20271.048,E2 -20271.048} C_VEL
LIN {X 0,Y 226.936,Z 493.93,A -85,B 0,C 180,E1 -20273.015,E2 -20273.015} C_VEL
LIN {X 0,Y 228.956,Z 482.628,A -85,B 0,C 180,E1 -20274.722,E2 -20274.722} C_VEL
LIN {X 0,Y 230.749,Z 470.924,A -85,B 0,C 180,E1 -20276.086,E2 -20276.086} C_VEL
LIN {X 0,Y 232.255,Z 459.014,A -85,B 0,C 180,E1 -20277.115,E2 -20277.115} C_VEL
LIN {X 0,Y 233.391,Z 445.947,A -85,B 0,C 180,E1 -20277.883,E2 -20277.883} C_VEL
LIN {X 0,Y 234.092,Z 427.287,A -85,B 0,C 180,E1 -20278.524,E2 -20278.524} C_VEL
LIN {X 0,Y 235.385,Z 387.668,A -85,B 0,C 180,E1 -20279.693,E2 -20279.693} C_VEL
LIN {X 0,Y 231.716,Z 355.856,A -85,B 0,C 180,E1 -20281.205,E2 -20281.205} C_VEL
LIN {X 0,Y 226.191,Z 341.079,A -85,B 0,C 180,E1 -20282.437,E2 -20282.437} C_VEL
LIN {X 0,Y 223.322,Z 334.029,A -85,B 0,C 180,E1 -20283.116,E2 -20283.116} C_VEL
LIN {X 0,Y 221.273,Z 324.751,A -85,B 0,C 180,E1 -20287.118,E2 -20287.118} C_VEL
LIN {X 0,Y 220.837,Z 322.976,A -85,B 0,C 180,E1 -20287.921,E2 -20287.921} C_VEL
LIN {X 0,Y 220.76,Z 322.987,A -85,B 0,C 180,E1 -20292.927,E2 -20292.927} C_VEL
LIN {X 0,Y 220.76,Z 322.986,A -85,B 0,C 180,E1 -20297.071,E2 -20297.071} C_VEL
LIN {X 0,Y 220.805,Z 322.983,A -85,B 0,C 180,E1 -20300.462,E2 -20300.462} C_VEL
LIN {X 0,Y 220.799,Z 322.983,A -85,B 0,C 180,E1 -20305.044,E2 -20305.044} C_VEL
LIN {X 0,Y 220.866,Z 322.975,A -85,B 0,C 180,E1 -20309.394,E2 -20309.394} C_VEL
LIN {X 0,Y 220.893,Z 322.97,A -85,B 0,C 180,E1 -20313.549,E2 -20313.549} C_VEL
LIN {X 0,Y 220.875,Z 322.97,A -85,B 0,C 180,E1 -20317.553,E2 -20317.553} C_VEL
LIN {X 0,Y 220.982,Z 322.955,A -85,B 0,C 180,E1 -20322.57,E2 -20322.57} C_VEL
LIN {X 0,Y 221.01,Z 322.943,A -85,B 0,C 180,E1 -20327.138,E2 -20327.138} C_VEL
LIN {X 0,Y 221.233,Z 322.917,A -85,B 0,C 180,E1 -20330.86,E2 -20330.86} C_VEL
LIN {X 0,Y 221.285,Z 322.918,A -85,B 0,C 180,E1 -20332.701,E2 -20332.701} C_VEL
LIN {X 0,Y 221.508,Z 322.875,A -85,B 0,C 180,E1 -20338.181,E2 -20338.181} C_VEL
LIN {X 0,Y 221.507,Z 322.885,A -85,B 0,C 180,E1 -20341.818,E2 -20341.818} C_VEL
LIN {X 0,Y 221.244,Z 322.921,A -85,B 0,C 180,E1 -20347.3,E2 -20347.3} C_VEL
LIN {X 0,Y 221.064,Z 322.934,A -85,B 0,C 180,E1 -20350.996,E2 -20350.996} C_VEL
LIN {X 0,Y 220.992,Z 322.956,A -85,B 0,C 180,E1 -20354.739,E2 -20354.739} C_VEL
LIN {X 0,Y 220.916,Z 322.954,A -85,B 0,C 180,E1 -20358.549,E2 -20358.549} C_VEL
LIN {X 0,Y 220.881,Z 322.964,A -85,B 0,C 180,E1 -20362.675,E2 -20362.675} C_VEL
LIN {X 0,Y 220.882,Z 322.966,A -85,B 0,C 180,E1 -20367.016,E2 -20367.016} C_VEL
LIN {X 0,Y 220.86,Z 322.957,A -85,B 0,C 180,E1 -20370.779,E2 -20370.779} C_VEL
LIN {X 0,Y 220.797,Z 322.98,A -85,B 0,C 180,E1 -20374.955,E2 -20374.955} C_VEL
LIN {X 0,Y 220.802,Z 322.968,A -85,B 0,C 180,E1 -20379.537,E2 -20379.537} C_VEL
LIN {X 0,Y 220.759,Z 322.981,A -85,B 0,C 180,E1 -20384.457,E2 -20384.457} C_VEL
LIN {X 0,Y 220.745,Z 322.985,A -85,B 0,C 180,E1 -20388.043,E2 -20388.043} C_VEL
LIN {X 0,Y 220.822,Z 322.973,A -85,B 0,C 180,E1 -20392.794,E2 -20392.794} C_VEL
LIN {X 0,Y 220.808,Z 322.98,A -85,B 0,C 180,E1 -20397.244,E2 -20397.244} C_VEL
LIN {X 0,Y 220.793,Z 322.98,A -85,B 0,C 180,E1 -20401.481,E2 -20401.481} C_VEL
LIN {X 0,Y 220.824,Z 322.978,A -85,B 0,C 180,E1 -20405.561,E2 -20405.561} C_VEL
LIN {X 0,Y 220.851,Z 322.974,A -85,B 0,C 180,E1 -20406.738,E2 -20406.738} C_VEL
LIN {X 0,Y 221.877,Z 325.871,A -85,B 0,C 180,E1 -20407.008,E2 -20407.008} C_VEL
LIN {X 0,Y 229.301,Z 340.282,A -85,B 0,C 180,E1 -20408.54,E2 -20408.54} C_VEL
LIN {X 0,Y 235.054,Z 355.469,A -85,B 0,C 180,E1 -20409.783,E2 -20409.783} C_VEL
LIN {X 0,Y 236.244,Z 358.623,A -85,B 0,C 180,E1 -20410.032,E2 -20410.032} C_VEL
LIN {X 0,Y 234.357,Z 417.587,A -85,B 0,C 180,E1 -20411.776,E2 -20411.776} C_VEL
LIN {X 0,Y 233.703,Z 431.998,A -85,B 0,C 180,E1 -20412.317,E2 -20412.317} C_VEL
LIN {X 0,Y 232.787,Z 444.262,A -85,B 0,C 180,E1 -20413.108,E2 -20413.108} C_VEL
LIN {X 0,Y 231.358,Z 457.721,A -85,B 0,C 180,E1 -20414.36,E2 -20414.36} C_VEL
LIN {X 0,Y 229.731,Z 467.987,A -85,B 0,C 180,E1 -20415.608,E2 -20415.608} C_VEL
LIN {X 0,Y 227.715,Z 478.91,A -85,B 0,C 180,E1 -20417.298,E2 -20417.298} C_VEL
LIN {X 0,Y 225.947,Z 488.727,A -85,B 0,C 180,E1 -20419.245,E2 -20419.245} C_VEL
LIN {X 0,Y 224.145,Z 497.668,A -85,B 0,C 180,E1 -20421.436,E2 -20421.436} C_VEL
LIN {X 0,Y 222.348,Z 506.402,A -85,B 0,C 180,E1 -20424.105,E2 -20424.105} C_VEL
LIN {X 0,Y 220.895,Z 513.382,A -85,B 0,C 180,E1 -20426.809,E2 -20426.809} C_VEL
LIN {X 0,Y 219.82,Z 519.763,A -85,B 0,C 180,E1 -20430.001,E2 -20430.001} C_VEL
LIN {X 0,Y 219.164,Z 523.977,A -85,B 0,C 180,E1 -20432.758,E2 -20432.758} C_VEL
LIN {X 0,Y 218.919,Z 527.22,A -85,B 0,C 180,E1 -20435.621,E2 -20435.621} C_VEL
LIN {X 0,Y 218.619,Z 528.72,A -85,B 0,C 180,E1 -20437.389,E2 -20437.389} C_VEL
LIN {X 0,Y 218.468,Z 529.874,A -85,B 0,C 180,E1 -20439.257,E2 -20439.257} C_VEL
LIN {X 0,Y 218.637,Z 530.938,A -85,B 0,C 180,E1 -20443.004,E2 -20443.004} C_VEL
LIN {X 0,Y 219.153,Z 530.675,A -85,B 0,C 180,E1 -20445.833,E2 -20445.833} C_VEL
LIN {X 0,Y 219.826,Z 529.502,A -85,B 0,C 180,E1 -20448.646,E2 -20448.646} C_VEL
LIN {X 0,Y 220.517,Z 528.195,A -85,B 0,C 180,E1 -20450.523,E2 -20450.523} C_VEL
LIN {X 0,Y 221.938,Z 525.393,A -85,B 0,C 180,E1 -20453.318,E2 -20453.318} C_VEL
LIN {X 0,Y 223.8,Z 521.521,A -85,B 0,C 180,E1 -20456.082,E2 -20456.082} C_VEL
LIN {X 0,Y 226.014,Z 516.464,A -85,B 0,C 180,E1 -20458.815,E2 -20458.815} C_VEL
LIN {X 0,Y 228.75,Z 510.049,A -85,B 0,C 180,E1 -20461.487,E2 -20461.487} C_VEL
LIN {X 0,Y 231.929,Z 501.948,A -85,B 0,C 180,E1 -20464.097,E2 -20464.097} C_VEL
LIN {X 0,Y 235.16,Z 493.067,A -85,B 0,C 180,E1 -20466.344,E2 -20466.344} C_VEL
LIN {X 0,Y 238.255,Z 483.445,A -85,B 0,C 180,E1 -20468.277,E2 -20468.277} C_VEL
LIN {X 0,Y 240.964,Z 473.231,A -85,B 0,C 180,E1 -20469.916,E2 -20469.916} C_VEL
LIN {X 0,Y 243.617,Z 461.676,A -85,B 0,C 180,E1 -20471.351,E2 -20471.351} C_VEL
LIN {X 0,Y 245.756,Z 449.586,A -85,B 0,C 180,E1 -20472.502,E2 -20472.502} C_VEL
LIN {X 0,Y 247.383,Z 436.797,A -85,B 0,C 180,E1 -20473.368,E2 -20473.368} C_VEL
LIN {X 0,Y 248.37,Z 425.398,A -85,B 0,C 180,E1 -20473.869,E2 -20473.869} C_VEL
LIN {X 0,Y 251.049,Z 374.889,A -85,B 0,C 180,E1 -20475.236,E2 -20475.236} C_VEL
LIN {X 0,Y 244.585,Z 361.006,A -85,B 0,C 180,E1 -20477.036,E2 -20477.036} C_VEL
LIN {X 0,Y 237.206,Z 347.581,A -85,B 0,C 180,E1 -20479.185,E2 -20479.185} C_VEL
LIN {X 0,Y 230.067,Z 336.77,A -85,B 0,C 180,E1 -20481.387,E2 -20481.387} C_VEL
LIN {X 0,Y 226.754,Z 332.219,A -85,B 0,C 180,E1 -20482.467,E2 -20482.467} C_VEL
LIN {X 0,Y 224.523,Z 329.098,A -85,B 0,C 180,E1 -20483.227,E2 -20483.227} C_VEL
LIN {X 0,Y 223.687,Z 327.807,A -85,B 0,C 180,E1 -20483.525,E2 -20483.525} C_VEL
LIN {X 0,Y 221.652,Z 325.513,A -85,B 0,C 180,E1 -20484.225,E2 -20484.225} C_VEL
LIN {X 0,Y 220.817,Z 322.971,A -85,B 0,C 180,E1 -20484.63,E2 -20484.63} C_VEL
LIN {X 0,Y 220.869,Z 322.955,A -85,B 0,C 180,E1 -20489.395,E2 -20489.395} C_VEL
LIN {X 0,Y 220.895,Z 322.955,A -85,B 0,C 180,E1 -20493.55,E2 -20493.55} C_VEL
LIN {X 0,Y 220.866,Z 322.961,A -85,B 0,C 180,E1 -20497.553,E2 -20497.553} C_VEL
LIN {X 0,Y 220.985,Z 322.957,A -85,B 0,C 180,E1 -20502.572,E2 -20502.572} C_VEL
LIN {X 0,Y 221.027,Z 322.954,A -85,B 0,C 180,E1 -20507.14,E2 -20507.14} C_VEL
LIN {X 0,Y 221.259,Z 322.923,A -85,B 0,C 180,E1 -20510.862,E2 -20510.862} C_VEL
LIN {X 0,Y 221.312,Z 322.908,A -85,B 0,C 180,E1 -20512.703,E2 -20512.703} C_VEL
LIN {X 0,Y 221.513,Z 322.879,A -85,B 0,C 180,E1 -20518.182,E2 -20518.182} C_VEL
LIN {X 0,Y 221.513,Z 322.88,A -85,B 0,C 180,E1 -20521.819,E2 -20521.819} C_VEL
LIN {X 0,Y 221.291,Z 322.904,A -85,B 0,C 180,E1 -20527.299,E2 -20527.299} C_VEL
LIN {X 0,Y 221.109,Z 322.93,A -85,B 0,C 180,E1 -20530.995,E2 -20530.995} C_VEL
LIN {X 0,Y 221.018,Z 322.941,A -85,B 0,C 180,E1 -20536.63,E2 -20536.63} C_VEL
LIN {X 0,Y 220.887,Z 322.958,A -85,B 0,C 180,E1 -20540.487,E2 -20540.487} C_VEL
LIN {X 0,Y 220.864,Z 322.963,A -85,B 0,C 180,E1 -20544.436,E2 -20544.436} C_VEL
LIN {X 0,Y 220.829,Z 322.968,A -85,B 0,C 180,E1 -20548.515,E2 -20548.515} C_VEL
LIN {X 0,Y 220.795,Z 322.973,A -85,B 0,C 180,E1 -20551.861,E2 -20551.861} C_VEL
LIN {X 0,Y 220.116,Z 323.058,A -85,B 0,C 180,E1 -20552.873,E2 -20552.873} C_VEL
LIN {X 0,Y 217.271,Z 323.42,A -85,B 0,C 180,E1 -20554.463,E2 -20554.463} C_VEL
LIN {X 0,Y 214.397,Z 323.771,A -85,B 0,C 180,E1 -20556.093,E2 -20556.093} C_VEL
LIN {X 0,Y 213.715,Z 323.855,A -85,B 0,C 180,E1 -20557.151,E2 -20557.151} C_VEL
LIN {X 0,Y 213.737,Z 323.91,A -85,B 0,C 180,E1 -20558.547,E2 -20558.547} C_VEL
LIN {X 0,Y 215.81,Z 330.745,A -85,B 0,C 180,E1 -20563.148,E2 -20563.148} C_VEL
LIN {X 0,Y 216.324,Z 332.219,A -85,B 0,C 180,E1 -20564.009,E2 -20564.009} C_VEL
LIN {X 0,Y 219.01,Z 336.651,A -85,B 0,C 180,E1 -20565.066,E2 -20565.066} C_VEL
LIN {X 0,Y 220.562,Z 338.927,A -85,B 0,C 180,E1 -20565.638,E2 -20565.638} C_VEL
LIN {X 0,Y 224.197,Z 344.875,A -85,B 0,C 180,E1 -20566.953,E2 -20566.953} C_VEL
LIN {X 0,Y 229.802,Z 354.518,A -85,B 0,C 180,E1 -20568.861,E2 -20568.861} C_VEL
LIN {X 0,Y 235.941,Z 366.541,A -85,B 0,C 180,E1 -20570.842,E2 -20570.842} C_VEL
LIN {X 0,Y 241.644,Z 379.068,A -85,B 0,C 180,E1 -20572.589,E2 -20572.589} C_VEL
LIN {X 0,Y 242.939,Z 382.636,A -85,B 0,C 180,E1 -20572.995,E2 -20572.995} C_VEL
LIN {X 0,Y 244.651,Z 394.833,A -85,B 0,C 180,E1 -20573.806,E2 -20573.806} C_VEL
LIN {X 0,Y 242.151,Z 442.572,A -85,B 0,C 180,E1 -20575.177,E2 -20575.177} C_VEL
LIN {X 0,Y 240.571,Z 456.292,A -85,B 0,C 180,E1 -20575.866,E2 -20575.866} C_VEL
LIN {X 0,Y 238.31,Z 469.033,A -85,B 0,C 180,E1 -20576.809,E2 -20576.809} C_VEL
LIN {X 0,Y 235.602,Z 480.815,A -85,B 0,C 180,E1 -20578.029,E2 -20578.029} C_VEL
LIN {X 0,Y 232.474,Z 492.165,A -85,B 0,C 180,E1 -20579.577,E2 -20579.577} C_VEL
LIN {X 0,Y 229.171,Z 502.422,A -85,B 0,C 180,E1 -20581.368,E2 -20581.368} C_VEL
LIN {X 0,Y 225.546,Z 512.465,A -85,B 0,C 180,E1 -20583.638,E2 -20583.638} C_VEL
LIN {X 0,Y 221.959,Z 521.311,A -85,B 0,C 180,E1 -20586.189,E2 -20586.189} C_VEL
LIN {X 0,Y 219.23,Z 528.247,A -85,B 0,C 180,E1 -20588.772,E2 -20588.772} C_VEL
LIN {X 0,Y 217.037,Z 533.27,A -85,B 0,C 180,E1 -20591.106,E2 -20591.106} C_VEL
LIN {X 0,Y 214.931,Z 537.984,A -85,B 0,C 180,E1 -20593.862,E2 -20593.862} C_VEL
LIN {X 0,Y 213.332,Z 541.608,A -85,B 0,C 180,E1 -20596.667,E2 -20596.667} C_VEL
LIN {X 0,Y 212.626,Z 543.495,A -85,B 0,C 180,E1 -20598.561,E2 -20598.561} C_VEL
LIN {X 0,Y 211.69,Z 545.959,A -85,B 0,C 180,E1 -20602.368,E2 -20602.368} C_VEL
LIN {X 0,Y 211.438,Z 546.881,A -85,B 0,C 180,E1 -20606.188,E2 -20606.188} C_VEL
LIN {X 0,Y 211.545,Z 546.729,A -85,B 0,C 180,E1 -20608.095,E2 -20608.095} C_VEL
LIN {X 0,Y 211.662,Z 546.171,A -85,B 0,C 180,E1 -20609.999,E2 -20609.999} C_VEL
LIN {X 0,Y 211.574,Z 545.208,A -85,B 0,C 180,E1 -20611.903,E2 -20611.903} C_VEL
LIN {X 0,Y 211.508,Z 543.167,A -85,B 0,C 180,E1 -20614.548,E2 -20614.548} C_VEL
LIN {X 0,Y 211.713,Z 539.717,A -85,B 0,C 180,E1 -20617.63,E2 -20617.63} C_VEL
LIN {X 0,Y 212.169,Z 535.377,A -85,B 0,C 180,E1 -20620.496,E2 -20620.496} C_VEL
LIN {X 0,Y 213.001,Z 529.824,A -85,B 0,C 180,E1 -20623.353,E2 -20623.353} C_VEL
LIN {X 0,Y 214.454,Z 522.891,A -85,B 0,C 180,E1 -20626.173,E2 -20626.173} C_VEL
LIN {X 0,Y 215.992,Z 515.8,A -85,B 0,C 180,E1 -20628.496,E2 -20628.496} C_VEL
LIN {X 0,Y 217.603,Z 507.206,A -85,B 0,C 180,E1 -20630.809,E2 -20630.809} C_VEL
LIN {X 0,Y 219.463,Z 497.771,A -85,B 0,C 180,E1 -20632.847,E2 -20632.847} C_VEL
LIN {X 0,Y 221.432,Z 487.508,A -85,B 0,C 180,E1 -20634.617,E2 -20634.617} C_VEL
LIN {X 0,Y 223.373,Z 476.299,A -85,B 0,C 180,E1 -20636.134,E2 -20636.134} C_VEL
LIN {X 0,Y 225.103,Z 463.767,A -85,B 0,C 180,E1 -20637.419,E2 -20637.419} C_VEL
LIN {X 0,Y 226.545,Z 450.372,A -85,B 0,C 180,E1 -20638.36,E2 -20638.36} C_VEL
LIN {X 0,Y 227.283,Z 437.163,A -85,B 0,C 180,E1 -20638.954,E2 -20638.954} C_VEL
LIN {X 0,Y 228.958,Z 388.42,A -85,B 0,C 180,E1 -20640.429,E2 -20640.429} C_VEL
LIN {X 0,Y 225.456,Z 357.411,A -85,B 0,C 180,E1 -20641.957,E2 -20641.957} C_VEL
LIN {X 0,Y 218.846,Z 340.548,A -85,B 0,C 180,E1 -20643.481,E2 -20643.481} C_VEL
LIN {X 0,Y 216.05,Z 333.732,A -85,B 0,C 180,E1 -20644.182,E2 -20644.182} C_VEL
LIN {X 0,Y 214.103,Z 325.251,A -85,B 0,C 180,E1 -20648.018,E2 -20648.018} C_VEL
LIN {X 0,Y 213.753,Z 323.86,A -85,B 0,C 180,E1 -20648.735,E2 -20648.735} C_VEL
LIN {X 0,Y 213.702,Z 323.865,A -85,B 0,C 180,E1 -20653.678,E2 -20653.678} C_VEL
LIN {X 0,Y 213.701,Z 323.868,A -85,B 0,C 180,E1 -20656.344,E2 -20656.344} C_VEL
LIN {X 0,Y 213.715,Z 323.864,A -85,B 0,C 180,E1 -20659.142,E2 -20659.142} C_VEL
LIN {X 0,Y 213.742,Z 323.863,A -85,B 0,C 180,E1 -20663.711,E2 -20663.711} C_VEL
LIN {X 0,Y 213.793,Z 323.856,A -85,B 0,C 180,E1 -20668.724,E2 -20668.724} C_VEL
LIN {X 0,Y 213.824,Z 323.851,A -85,B 0,C 180,E1 -20672.602,E2 -20672.602} C_VEL
LIN {X 0,Y 213.85,Z 323.85,A -85,B 0,C 180,E1 -20676.952,E2 -20676.952} C_VEL
LIN {X 0,Y 213.941,Z 323.833,A -85,B 0,C 180,E1 -20682.803,E2 -20682.803} C_VEL
LIN {X 0,Y 213.951,Z 323.827,A -85,B 0,C 180,E1 -20686.706,E2 -20686.706} C_VEL
LIN {X 0,Y 214.164,Z 323.796,A -85,B 0,C 180,E1 -20690.556,E2 -20690.556} C_VEL
LIN {X 0,Y 214.223,Z 323.797,A -85,B 0,C 180,E1 -20692.459,E2 -20692.459} C_VEL
LIN {X 0,Y 214.441,Z 323.755,A -85,B 0,C 180,E1 -20698.121,E2 -20698.121} C_VEL
LIN {X 0,Y 214.542,Z 323.742,A -85,B 0,C 180,E1 -20700,E2 -20700} C_VEL
LIN {X 0,Y 214.44,Z 323.766,A -85,B 0,C 180,E1 -20701.878,E2 -20701.878} C_VEL
LIN {X 0,Y 214.185,Z 323.796,A -85,B 0,C 180,E1 -20707.542,E2 -20707.542} C_VEL
LIN {X 0,Y 213.995,Z 323.814,A -85,B 0,C 180,E1 -20711.364,E2 -20711.364} C_VEL
LIN {X 0,Y 213.93,Z 323.836,A -85,B 0,C 180,E1 -20715.237,E2 -20715.237} C_VEL
LIN {X 0,Y 213.832,Z 323.834,A -85,B 0,C 180,E1 -20719.188,E2 -20719.188} C_VEL
LIN {X 0,Y 213.807,Z 323.848,A -85,B 0,C 180,E1 -20723.231,E2 -20723.231} C_VEL
LIN {X 0,Y 213.826,Z 323.844,A -85,B 0,C 180,E1 -20727.45,E2 -20727.45} C_VEL
LIN {X 0,Y 213.773,Z 323.845,A -85,B 0,C 180,E1 -20731.736,E2 -20731.736} C_VEL
LIN {X 0,Y 213.74,Z 323.857,A -85,B 0,C 180,E1 -20736.289,E2 -20736.289} C_VEL
LIN {X 0,Y 213.707,Z 323.86,A -85,B 0,C 180,E1 -20741.126,E2 -20741.126} C_VEL
LIN {X 0,Y 213.699,Z 323.861,A -85,B 0,C 180,E1 -20743.68,E2 -20743.68} C_VEL
LIN {X 0,Y 213.698,Z 323.852,A -85,B 0,C 180,E1 -20746.346,E2 -20746.346} C_VEL
LIN {X 0,Y 213.703,Z 323.857,A -85,B 0,C 180,E1 -20751.33,E2 -20751.33} C_VEL
LIN {X 0,Y 213.753,Z 323.858,A -85,B 0,C 180,E1 -20756.018,E2 -20756.018} C_VEL
LIN {X 0,Y 213.744,Z 323.853,A -85,B 0,C 180,E1 -20760.449,E2 -20760.449} C_VEL
LIN {X 0,Y 213.76,Z 323.855,A -85,B 0,C 180,E1 -20764.697,E2 -20764.697} C_VEL
LIN {X 0,Y 213.8,Z 323.852,A -85,B 0,C 180,E1 -20765.705,E2 -20765.705} C_VEL
LIN {X 0,Y 214.892,Z 326.837,A -85,B 0,C 180,E1 -20766.003,E2 -20766.003} C_VEL
LIN {X 0,Y 222.17,Z 340.669,A -85,B 0,C 180,E1 -20767.587,E2 -20767.587} C_VEL
LIN {X 0,Y 226.877,Z 351.914,A -85,B 0,C 180,E1 -20768.628,E2 -20768.628} C_VEL
LIN {X 0,Y 229.966,Z 361.187,A -85,B 0,C 180,E1 -20769.349,E2 -20769.349} C_VEL
LIN {X 0,Y 227.485,Z 427.705,A -85,B 0,C 180,E1 -20771.386,E2 -20771.386} C_VEL
LIN {X 0,Y 226.58,Z 441.192,A -85,B 0,C 180,E1 -20772.164,E2 -20772.164} C_VEL
LIN {X 0,Y 225.335,Z 453.654,A -85,B 0,C 180,E1 -20773.233,E2 -20773.233} C_VEL
LIN {X 0,Y 223.833,Z 464.79,A -85,B 0,C 180,E1 -20774.522,E2 -20774.522} C_VEL
LIN {X 0,Y 221.794,Z 475.129,A -85,B 0,C 180,E1 -20776.019,E2 -20776.019} C_VEL
LIN {X 0,Y 219.828,Z 485.738,A -85,B 0,C 180,E1 -20778.007,E2 -20778.007} C_VEL
LIN {X 0,Y 217.831,Z 495.311,A -85,B 0,C 180,E1 -20780.249,E2 -20780.249} C_VEL
LIN {X 0,Y 216.189,Z 503.149,A -85,B 0,C 180,E1 -20782.529,E2 -20782.529} C_VEL
LIN {X 0,Y 214.492,Z 510.817,A -85,B 0,C 180,E1 -20785.302,E2 -20785.302} C_VEL
LIN {X 0,Y 213.296,Z 516.966,A -85,B 0,C 180,E1 -20788.112,E2 -20788.112} C_VEL
LIN {X 0,Y 212.376,Z 521.861,A -85,B 0,C 180,E1 -20790.949,E2 -20790.949} C_VEL
LIN {X 0,Y 211.963,Z 525.63,A -85,B 0,C 180,E1 -20793.803,E2 -20793.803} C_VEL
LIN {X 0,Y 211.808,Z 527.581,A -85,B 0,C 180,E1 -20795.713,E2 -20795.713} C_VEL
LIN {X 0,Y 211.495,Z 529.134,A -85,B 0,C 180,E1 -20797.639,E2 -20797.639} C_VEL
LIN {X 0,Y 211.377,Z 530.225,A -85,B 0,C 180,E1 -20799.57,E2 -20799.57} C_VEL
LIN {X 0,Y 211.619,Z 531.222,A -85,B 0,C 180,E1 -20803.443,E2 -20803.443} C_VEL
LIN {X 0,Y 212.108,Z 530.962,A -85,B 0,C 180,E1 -20806.079,E2 -20806.079} C_VEL
LIN {X 0,Y 212.919,Z 529.653,A -85,B 0,C 180,E1 -20809.274,E2 -20809.274} C_VEL
LIN {X 0,Y 213.706,Z 528.311,A -85,B 0,C 180,E1 -20811.208,E2 -20811.208} C_VEL
LIN {X 0,Y 215.08,Z 525.753,A -85,B 0,C 180,E1 -20813.804,E2 -20813.804} C_VEL
LIN {X 0,Y 217.232,Z 521.487,A -85,B 0,C 180,E1 -20816.933,E2 -20816.933} C_VEL
LIN {X 0,Y 219.615,Z 516.383,A -85,B 0,C 180,E1 -20819.715,E2 -20819.715} C_VEL
LIN {X 0,Y 222.559,Z 509.795,A -85,B 0,C 180,E1 -20822.468,E2 -20822.468} C_VEL
LIN {X 0,Y 225.94,Z 501.584,A -85,B 0,C 180,E1 -20825.132,E2 -20825.132} C_VEL
LIN {X 0,Y 229.331,Z 492.605,A -85,B 0,C 180,E1 -20827.414,E2 -20827.414} C_VEL
LIN {X 0,Y 232.553,Z 482.718,A -85,B 0,C 180,E1 -20829.394,E2 -20829.394} C_VEL
LIN {X 0,Y 235.74,Z 471.119,A -85,B 0,C 180,E1 -20831.214,E2 -20831.214} C_VEL
LIN {X 0,Y 238.132,Z 460.891,A -85,B 0,C 180,E1 -20832.454,E2 -20832.454} C_VEL
LIN {X 0,Y 240.233,Z 449.066,A -85,B 0,C 180,E1 -20833.577,E2 -20833.577} C_VEL
LIN {X 0,Y 241.875,Z 436.022,A -85,B 0,C 180,E1 -20834.452,E2 -20834.452} C_VEL
LIN {X 0,Y 243.006,Z 423.689,A -85,B 0,C 180,E1 -20834.952,E2 -20834.952} C_VEL
LIN {X 0,Y 245.468,Z 376.991,A -85,B 0,C 180,E1 -20836.244,E2 -20836.244} C_VEL
LIN {X 0,Y 238.976,Z 363.203,A -85,B 0,C 180,E1 -20838.148,E2 -20838.148} C_VEL
LIN {X 0,Y 232.699,Z 351.827,A -85,B 0,C 180,E1 -20840.075,E2 -20840.075} C_VEL
LIN {X 0,Y 226.013,Z 341.676,A -85,B 0,C 180,E1 -20842.235,E2 -20842.235} C_VEL
LIN {X 0,Y 222.845,Z 337.3,A -85,B 0,C 180,E1 -20843.315,E2 -20843.315} C_VEL
LIN {X 0,Y 220.095,Z 333.353,A -85,B 0,C 180,E1 -20844.307,E2 -20844.307} C_VEL
LIN {X 0,Y 217.721,Z 330.128,A -85,B 0,C 180,E1 -20845.193,E2 -20845.193} C_VEL
LIN {X 0,Y 216.979,Z 328.956,A -85,B 0,C 180,E1 -20845.486,E2 -20845.486} C_VEL
LIN {X 0,Y 214.725,Z 326.652,A -85,B 0,C 180,E1 -20846.333,E2 -20846.333} C_VEL
LIN {X 0,Y 213.76,Z 323.849,A -85,B 0,C 180,E1 -20846.831,E2 -20846.831} C_VEL
LIN {X 0,Y 213.781,Z 323.845,A -85,B 0,C 180,E1 -20850.455,E2 -20850.455} C_VEL
LIN {X 0,Y 213.8,Z 323.847,A -85,B 0,C 180,E1 -20854.702,E2 -20854.702} C_VEL
LIN {X 0,Y 213.805,Z 323.85,A -85,B 0,C 180,E1 -20858.803,E2 -20858.803} C_VEL
LIN {X 0,Y 213.945,Z 323.835,A -85,B 0,C 180,E1 -20862.804,E2 -20862.804} C_VEL
LIN {X 0,Y 213.982,Z 323.831,A -85,B 0,C 180,E1 -20866.709,E2 -20866.709} C_VEL
LIN {X 0,Y 214.198,Z 323.8,A -85,B 0,C 180,E1 -20870.558,E2 -20870.558} C_VEL
LIN {X 0,Y 214.249,Z 323.79,A -85,B 0,C 180,E1 -20872.461,E2 -20872.461} C_VEL
LIN {X 0,Y 214.447,Z 323.759,A -85,B 0,C 180,E1 -20878.122,E2 -20878.122} C_VEL
LIN {X 0,Y 214.548,Z 323.757,A -85,B 0,C 180,E1 -20880,E2 -20880} C_VEL
LIN {X 0,Y 214.446,Z 323.76,A -85,B 0,C 180,E1 -20881.878,E2 -20881.878} C_VEL
LIN {X 0,Y 214.229,Z 323.784,A -85,B 0,C 180,E1 -20887.541,E2 -20887.541} C_VEL
LIN {X 0,Y 214.025,Z 323.81,A -85,B 0,C 180,E1 -20891.363,E2 -20891.363} C_VEL
LIN {X 0,Y 213.935,Z 323.826,A -85,B 0,C 180,E1 -20895.237,E2 -20895.237} C_VEL
LIN {X 0,Y 213.838,Z 323.843,A -85,B 0,C 180,E1 -20899.188,E2 -20899.188} C_VEL
LIN {X 0,Y 213.813,Z 323.849,A -85,B 0,C 180,E1 -20903.231,E2 -20903.231} C_VEL
LIN {X 0,Y 213.831,Z 323.845,A -85,B 0,C 180,E1 -20907.45,E2 -20907.45} C_VEL
LIN {X 0,Y 213.763,Z 323.85,A -85,B 0,C 180,E1 -20911.825,E2 -20911.825} C_VEL
LIN {X 0,Y 213.746,Z 323.851,A -85,B 0,C 180,E1 -20916.288,E2 -20916.288} C_VEL
LIN {X 0,Y 213.715,Z 323.855,A -85,B 0,C 180,E1 -20917.151,E2 -20917.151} C_VEL
LIN {X 0,Y 213.254,Z 324.368,A -85,B 0,C 180,E1 -20918.049,E2 -20918.049} C_VEL
LIN {X 0,Y 211.723,Z 326.273,A -85,B 0,C 180,E1 -20919.193,E2 -20919.193} C_VEL
LIN {X 0,Y 209.655,Z 330.126,A -85,B 0,C 180,E1 -20920.677,E2 -20920.677} C_VEL
LIN {X 0,Y 209.542,Z 332.866,A -85,B 0,C 180,E1 -20921.617,E2 -20921.617} C_VEL
LIN {X 0,Y 210.269,Z 334.231,A -85,B 0,C 180,E1 -20922.094,E2 -20922.094} C_VEL
LIN {X 0,Y 213.092,Z 338.137,A -85,B 0,C 180,E1 -20923.267,E2 -20923.267} C_VEL
LIN {X 0,Y 217.375,Z 344.993,A -85,B 0,C 180,E1 -20924.982,E2 -20924.982} C_VEL
LIN {X 0,Y 221.015,Z 351.028,A -85,B 0,C 180,E1 -20926.351,E2 -20926.351} C_VEL
LIN {X 0,Y 227.047,Z 361.722,A -85,B 0,C 180,E1 -20928.478,E2 -20928.478} C_VEL
LIN {X 0,Y 234.261,Z 376.751,A -85,B 0,C 180,E1 -20930.879,E2 -20930.879} C_VEL
LIN {X 0,Y 237.796,Z 385.477,A -85,B 0,C 180,E1 -20932.023,E2 -20932.023} C_VEL
LIN {X 0,Y 239.224,Z 395.703,A -85,B 0,C 180,E1 -20932.733,E2 -20932.733} C_VEL
LIN {X 0,Y 236.693,Z 442.197,A -85,B 0,C 180,E1 -20934.09,E2 -20934.09} C_VEL
LIN {X 0,Y 235.091,Z 455.709,A -85,B 0,C 180,E1 -20934.771,E2 -20934.771} C_VEL
LIN {X 0,Y 232.889,Z 467.902,A -85,B 0,C 180,E1 -20935.671,E2 -20935.671} C_VEL
LIN {X 0,Y 230.019,Z 479.924,A -85,B 0,C 180,E1 -20936.896,E2 -20936.896} C_VEL
LIN {X 0,Y 226.819,Z 491.38,A -85,B 0,C 180,E1 -20938.474,E2 -20938.474} C_VEL
LIN {X 0,Y 223.361,Z 501.726,A -85,B 0,C 180,E1 -20940.292,E2 -20940.292} C_VEL
LIN {X 0,Y 219.885,Z 511.054,A -85,B 0,C 180,E1 -20942.39,E2 -20942.39} C_VEL
LIN {X 0,Y 216.084,Z 520.088,A -85,B 0,C 180,E1 -20944.987,E2 -20944.987} C_VEL
LIN {X 0,Y 212.93,Z 527.473,A -85,B 0,C 180,E1 -20947.731,E2 -20947.731} C_VEL
LIN {X 0,Y 210.301,Z 533.268,A -85,B 0,C 180,E1 -20950.476,E2 -20950.476} C_VEL
LIN {X 0,Y 208.114,Z 537.926,A -85,B 0,C 180,E1 -20953.318,E2 -20953.318} C_VEL
LIN {X 0,Y 206.385,Z 541.497,A -85,B 0,C 180,E1 -20956.209,E2 -20956.209} C_VEL
LIN {X 0,Y 205.625,Z 543.343,A -85,B 0,C 180,E1 -20958.166,E2 -20958.166} C_VEL
LIN {X 0,Y 204.642,Z 545.752,A -85,B 0,C 180,E1 -20962.104,E2 -20962.104} C_VEL
LIN {X 0,Y 204.338,Z 546.618,A -85,B 0,C 180,E1 -20966.055,E2 -20966.055} C_VEL
LIN {X 0,Y 204.46,Z 546.43,A -85,B 0,C 180,E1 -20968.029,E2 -20968.029} C_VEL
LIN {X 0,Y 204.575,Z 545.848,A -85,B 0,C 180,E1 -20969.999,E2 -20969.999} C_VEL
LIN {X 0,Y 204.471,Z 544.861,A -85,B 0,C 180,E1 -20971.969,E2 -20971.969} C_VEL
LIN {X 0,Y 204.412,Z 543.063,A -85,B 0,C 180,E1 -20974.386,E2 -20974.386} C_VEL
LIN {X 0,Y 204.655,Z 539.269,A -85,B 0,C 180,E1 -20977.894,E2 -20977.894} C_VEL
LIN {X 0,Y 205.141,Z 534.873,A -85,B 0,C 180,E1 -20980.86,E2 -20980.86} C_VEL
LIN {X 0,Y 206.06,Z 529.262,A -85,B 0,C 180,E1 -20983.812,E2 -20983.812} C_VEL
LIN {X 0,Y 207.596,Z 522.258,A -85,B 0,C 180,E1 -20986.723,E2 -20986.723} C_VEL
LIN {X 0,Y 209.513,Z 513.447,A -85,B 0,C 180,E1 -20989.599,E2 -20989.599} C_VEL
LIN {X 0,Y 211.445,Z 503.391,A -85,B 0,C 180,E1 -20992.214,E2 -20992.214} C_VEL
LIN {X 0,Y 213.649,Z 493.191,A -85,B 0,C 180,E1 -20994.279,E2 -20994.279} C_VEL
LIN {X 0,Y 215.795,Z 481.836,A -85,B 0,C 180,E1 -20996.082,E2 -20996.082} C_VEL
LIN {X 0,Y 217.692,Z 470.056,A -85,B 0,C 180,E1 -20997.52,E2 -20997.52} C_VEL
LIN {X 0,Y 219.379,Z 457.224,A -85,B 0,C 180,E1 -20998.654,E2 -20998.654} C_VEL
LIN {X 0,Y 220.585,Z 443.485,A -85,B 0,C 180,E1 -20999.461,E2 -20999.461} C_VEL
LIN {X 0,Y 221.95,Z 409.585,A -85,B 0,C 180,E1 -21000.561,E2 -21000.561} C_VEL
LIN {X 0,Y 222.545,Z 388.948,A -85,B 0,C 180,E1 -21001.219,E2 -21001.219} C_VEL
LIN {X 0,Y 219.432,Z 360.26,A -85,B 0,C 180,E1 -21002.675,E2 -21002.675} C_VEL
LIN {X 0,Y 214.469,Z 346.977,A -85,B 0,C 180,E1 -21003.888,E2 -21003.888} C_VEL
LIN {X 0,Y 208.796,Z 333.456,A -85,B 0,C 180,E1 -21005.32,E2 -21005.32} C_VEL
LIN {X 0,Y 206.748,Z 324.732,A -85,B 0,C 180,E1 -21009.543,E2 -21009.543} C_VEL
LIN {X 0,Y 206.63,Z 324.747,A -85,B 0,C 180,E1 -21014.416,E2 -21014.416} C_VEL
LIN {X 0,Y 206.639,Z 324.748,A -85,B 0,C 180,E1 -21018.437,E2 -21018.437} C_VEL
LIN {X 0,Y 206.678,Z 324.742,A -85,B 0,C 180,E1 -21022.259,E2 -21022.259} C_VEL
LIN {X 0,Y 206.7,Z 324.74,A -85,B 0,C 180,E1 -21027.042,E2 -21027.042} C_VEL
LIN {X 0,Y 206.764,Z 324.729,A -85,B 0,C 180,E1 -21032.096,E2 -21032.096} C_VEL
LIN {X 0,Y 206.783,Z 324.728,A -85,B 0,C 180,E1 -21036.583,E2 -21036.583} C_VEL
LIN {X 0,Y 206.871,Z 324.712,A -85,B 0,C 180,E1 -21042.196,E2 -21042.196} C_VEL
LIN {X 0,Y 206.893,Z 324.707,A -85,B 0,C 180,E1 -21046.244,E2 -21046.244} C_VEL
LIN {X 0,Y 207.102,Z 324.673,A -85,B 0,C 180,E1 -21050.231,E2 -21050.231} C_VEL
LIN {X 0,Y 207.164,Z 324.677,A -85,B 0,C 180,E1 -21052.201,E2 -21052.201} C_VEL
LIN {X 0,Y 207.378,Z 324.634,A -85,B 0,C 180,E1 -21058.057,E2 -21058.057} C_VEL
LIN {X 0,Y 207.508,Z 324.617,A -85,B 0,C 180,E1 -21060,E2 -21060} C_VEL
LIN {X 0,Y 207.376,Z 324.645,A -85,B 0,C 180,E1 -21061.942,E2 -21061.942} C_VEL
LIN {X 0,Y 207.128,Z 324.672,A -85,B 0,C 180,E1 -21067.8,E2 -21067.8} C_VEL
LIN {X 0,Y 206.921,Z 324.696,A -85,B 0,C 180,E1 -21071.758,E2 -21071.758} C_VEL
LIN {X 0,Y 206.864,Z 324.717,A -85,B 0,C 180,E1 -21075.771,E2 -21075.771} C_VEL
LIN {X 0,Y 206.759,Z 324.71,A -85,B 0,C 180,E1 -21079.871,E2 -21079.871} C_VEL
LIN {X 0,Y 206.743,Z 324.729,A -85,B 0,C 180,E1 -21084.074,E2 -21084.074} C_VEL
LIN {X 0,Y 206.741,Z 324.72,A -85,B 0,C 180,E1 -21088.419,E2 -21088.419} C_VEL
LIN {X 0,Y 206.699,Z 324.733,A -85,B 0,C 180,E1 -21092.957,E2 -21092.957} C_VEL
LIN {X 0,Y 206.676,Z 324.728,A -85,B 0,C 180,E1 -21097.74,E2 -21097.74} C_VEL
LIN {X 0,Y 206.637,Z 324.742,A -85,B 0,C 180,E1 -21101.563,E2 -21101.563} C_VEL
LIN {X 0,Y 206.626,Z 324.732,A -85,B 0,C 180,E1 -21105.583,E2 -21105.583} C_VEL
LIN {X 0,Y 206.644,Z 324.742,A -85,B 0,C 180,E1 -21109.746,E2 -21109.746} C_VEL
LIN {X 0,Y 206.696,Z 324.738,A -85,B 0,C 180,E1 -21114.689,E2 -21114.689} C_VEL
LIN {X 0,Y 206.691,Z 324.733,A -85,B 0,C 180,E1 -21119.335,E2 -21119.335} C_VEL
LIN {X 0,Y 206.723,Z 324.732,A -85,B 0,C 180,E1 -21124.232,E2 -21124.232} C_VEL
LIN {X 0,Y 206.727,Z 324.731,A -85,B 0,C 180,E1 -21124.565,E2 -21124.565} C_VEL
LIN {X 0,Y 207.953,Z 327.935,A -85,B 0,C 180,E1 -21124.934,E2 -21124.934} C_VEL
LIN {X 0,Y 210.777,Z 332.985,A -85,B 0,C 180,E1 -21125.593,E2 -21125.593} C_VEL
LIN {X 0,Y 218.201,Z 347.68,A -85,B 0,C 180,E1 -21127.279,E2 -21127.279} C_VEL
LIN {X 0,Y 223.563,Z 362.23,A -85,B 0,C 180,E1 -21128.553,E2 -21128.553} C_VEL
LIN {X 0,Y 221.026,Z 428.557,A -85,B 0,C 180,E1 -21130.653,E2 -21130.653} C_VEL
LIN {X 0,Y 220.034,Z 442.452,A -85,B 0,C 180,E1 -21131.495,E2 -21131.495} C_VEL
LIN {X 0,Y 218.746,Z 454.608,A -85,B 0,C 180,E1 -21132.591,E2 -21132.591} C_VEL
LIN {X 0,Y 217.028,Z 466.363,A -85,B 0,C 180,E1 -21134.024,E2 -21134.024} C_VEL
LIN {X 0,Y 214.904,Z 476.468,A -85,B 0,C 180,E1 -21135.561,E2 -21135.561} C_VEL
LIN {X 0,Y 212.945,Z 486.882,A -85,B 0,C 180,E1 -21137.613,E2 -21137.613} C_VEL
LIN {X 0,Y 210.873,Z 496.295,A -85,B 0,C 180,E1 -21139.924,E2 -21139.924} C_VEL
LIN {X 0,Y 208.862,Z 505.349,A -85,B 0,C 180,E1 -21142.752,E2 -21142.752} C_VEL
LIN {X 0,Y 207.175,Z 512.659,A -85,B 0,C 180,E1 -21145.623,E2 -21145.623} C_VEL
LIN {X 0,Y 206.208,Z 517.605,A -85,B 0,C 180,E1 -21148.048,E2 -21148.048} C_VEL
LIN {X 0,Y 205.265,Z 522.422,A -85,B 0,C 180,E1 -21150.982,E2 -21150.982} C_VEL
LIN {X 0,Y 204.866,Z 526.116,A -85,B 0,C 180,E1 -21153.935,E2 -21153.935} C_VEL
LIN {X 0,Y 204.662,Z 528.036,A -85,B 0,C 180,E1 -21155.914,E2 -21155.914} C_VEL
LIN {X 0,Y 204.381,Z 529.526,A -85,B 0,C 180,E1 -21157.907,E2 -21157.907} C_VEL
LIN {X 0,Y 204.314,Z 531.238,A -85,B 0,C 180,E1 -21161.911,E2 -21161.911} C_VEL
LIN {X 0,Y 204.582,Z 531.508,A -85,B 0,C 180,E1 -21163.915,E2 -21163.915} C_VEL
LIN {X 0,Y 205.063,Z 531.251,A -85,B 0,C 180,E1 -21166.338,E2 -21166.338} C_VEL
LIN {X 0,Y 206.063,Z 529.803,A -85,B 0,C 180,E1 -21169.942,E2 -21169.942} C_VEL
LIN {X 0,Y 206.909,Z 528.419,A -85,B 0,C 180,E1 -21171.94,E2 -21171.94} C_VEL
LIN {X 0,Y 208.256,Z 526.101,A -85,B 0,C 180,E1 -21174.334,E2 -21174.334} C_VEL
LIN {X 0,Y 210.753,Z 521.445,A -85,B 0,C 180,E1 -21177.831,E2 -21177.831} C_VEL
LIN {X 0,Y 213.176,Z 516.512,A -85,B 0,C 180,E1 -21180.558,E2 -21180.558} C_VEL
LIN {X 0,Y 216.438,Z 509.543,A -85,B 0,C 180,E1 -21183.506,E2 -21183.506} C_VEL
LIN {X 0,Y 220.003,Z 501.226,A -85,B 0,C 180,E1 -21186.227,E2 -21186.227} C_VEL
LIN {X 0,Y 223.488,Z 492.376,A -85,B 0,C 180,E1 -21188.483,E2 -21188.483} C_VEL
LIN {X 0,Y 226.972,Z 482.004,A -85,B 0,C 180,E1 -21190.561,E2 -21190.561} C_VEL
LIN {X 0,Y 229.991,Z 471.363,A -85,B 0,C 180,E1 -21192.243,E2 -21192.243} C_VEL
LIN {X 0,Y 232.784,Z 459.552,A -85,B 0,C 180,E1 -21193.682,E2 -21193.682} C_VEL
LIN {X 0,Y 234.998,Z 447.158,A -85,B 0,C 180,E1 -21194.804,E2 -21194.804} C_VEL
LIN {X 0,Y 236.63,Z 434.001,A -85,B 0,C 180,E1 -21195.648,E2 -21195.648} C_VEL
LIN {X 0,Y 237.755,Z 421.234,A -85,B 0,C 180,E1 -21196.108,E2 -21196.108} C_VEL
LIN {X 0,Y 240.011,Z 379.286,A -85,B 0,C 180,E1 -21197.283,E2 -21197.283} C_VEL
LIN {X 0,Y 233.825,Z 366.276,A -85,B 0,C 180,E1 -21199.195,E2 -21199.195} C_VEL
LIN {X 0,Y 228.648,Z 356.677,A -85,B 0,C 180,E1 -21200.871,E2 -21200.871} C_VEL
LIN {X 0,Y 222.407,Z 347.066,A -85,B 0,C 180,E1 -21202.978,E2 -21202.978} C_VEL
LIN {X 0,Y 216.291,Z 338.456,A -85,B 0,C 180,E1 -21205.219,E2 -21205.219} C_VEL
LIN {X 0,Y 213.489,Z 334.591,A -85,B 0,C 180,E1 -21206.325,E2 -21206.325} C_VEL
LIN {X 0,Y 211.063,Z 331.525,A -85,B 0,C 180,E1 -21207.313,E2 -21207.313} C_VEL
LIN {X 0,Y 210.275,Z 330.007,A -85,B 0,C 180,E1 -21207.672,E2 -21207.672} C_VEL
LIN {X 0,Y 208.029,Z 327.973,A -85,B 0,C 180,E1 -21208.598,E2 -21208.598} C_VEL
LIN {X 0,Y 206.935,Z 325.758,A -85,B 0,C 180,E1 -21209.135,E2 -21209.135} C_VEL
LIN {X 0,Y 206.725,Z 324.716,A -85,B 0,C 180,E1 -21209.34,E2 -21209.34} C_VEL
LIN {X 0,Y 206.732,Z 324.72,A -85,B 0,C 180,E1 -21213.772,E2 -21213.772} C_VEL
LIN {X 0,Y 206.74,Z 324.725,A -85,B 0,C 180,E1 -21218.042,E2 -21218.042} C_VEL
LIN {X 0,Y 206.874,Z 324.713,A -85,B 0,C 180,E1 -21222.197,E2 -21222.197} C_VEL
LIN {X 0,Y 206.915,Z 324.707,A -85,B 0,C 180,E1 -21226.246,E2 -21226.246} C_VEL
LIN {X 0,Y 207.134,Z 324.677,A -85,B 0,C 180,E1 -21230.233,E2 -21230.233} C_VEL
LIN {X 0,Y 207.19,Z 324.671,A -85,B 0,C 180,E1 -21232.202,E2 -21232.202} C_VEL
LIN {X 0,Y 207.383,Z 324.639,A -85,B 0,C 180,E1 -21238.058,E2 -21238.058} C_VEL
LIN {X 0,Y 207.513,Z 324.633,A -85,B 0,C 180,E1 -21240,E2 -21240} C_VEL
LIN {X 0,Y 207.383,Z 324.639,A -85,B 0,C 180,E1 -21241.942,E2 -21241.942} C_VEL
LIN {X 0,Y 207.17,Z 324.664,A -85,B 0,C 180,E1 -21247.799,E2 -21247.799} C_VEL
LIN {X 0,Y 206.945,Z 324.691,A -85,B 0,C 180,E1 -21251.758,E2 -21251.758} C_VEL
LIN {X 0,Y 206.868,Z 324.703,A -85,B 0,C 180,E1 -21255.771,E2 -21255.771} C_VEL
LIN {X 0,Y 206.765,Z 324.718,A -85,B 0,C 180,E1 -21259.871,E2 -21259.871} C_VEL
LIN {X 0,Y 206.749,Z 324.722,A -85,B 0,C 180,E1 -21264.074,E2 -21264.074} C_VEL
LIN {X 0,Y 206.739,Z 324.723,A -85,B 0,C 180,E1 -21268.42,E2 -21268.42} C_VEL
LIN {X 0,Y 206.701,Z 324.728,A -85,B 0,C 180,E1 -21272.958,E2 -21272.958} C_VEL
LIN {X 0,Y 206.73,Z 324.85,A -85,B 0,C 180,E1 -21276.508,E2 -21276.508} C_VEL
LIN {X 0,Y 208.862,Z 331.603,A -85,B 0,C 180,E1 -21281.447,E2 -21281.447} C_VEL
LIN {X 0,Y 210.269,Z 334.231,A -85,B 0,C 180,E1 -21282.094,E2 -21282.094} C_VEL
LIN {X 0,Y 211.899,Z 336.696,A -85,B 0,C 180,E1 -21282.789,E2 -21282.789} C_VEL
LIN {X 0,Y 213.742,Z 341.321,A -85,B 0,C 180,E1 -21283.647,E2 -21283.647} C_VEL
LIN {X 0,Y 217.43,Z 355.343,A -85,B 0,C 180,E1 -21285.512,E2 -21285.512} C_VEL
LIN {X 0,Y 219.491,Z 360.031,A -85,B 0,C 180,E1 -21286.344,E2 -21286.344} C_VEL
LIN {X 0,Y 224.942,Z 370.483,A -85,B 0,C 180,E1 -21288.325,E2 -21288.325} C_VEL
LIN {X 0,Y 231.243,Z 384.368,A -85,B 0,C 180,E1 -21290.496,E2 -21290.496} C_VEL
LIN {X 0,Y 232.766,Z 388.396,A -85,B 0,C 180,E1 -21291.019,E2 -21291.019} C_VEL
LIN {X 0,Y 233.884,Z 396.886,A -85,B 0,C 180,E1 -21291.623,E2 -21291.623} C_VEL
LIN {X 0,Y 231.351,Z 441.611,A -85,B 0,C 180,E1 -21292.943,E2 -21292.943} C_VEL
LIN {X 0,Y 229.726,Z 454.966,A -85,B 0,C 180,E1 -21293.614,E2 -21293.614} C_VEL
LIN {X 0,Y 227.329,Z 467.86,A -85,B 0,C 180,E1 -21294.573,E2 -21294.573} C_VEL
LIN {X 0,Y 224.548,Z 479.032,A -85,B 0,C 180,E1 -21295.71,E2 -21295.71} C_VEL
LIN {X 0,Y 221.233,Z 490.6,A -85,B 0,C 180,E1 -21297.313,E2 -21297.313} C_VEL
LIN {X 0,Y 217.646,Z 501.033,A -85,B 0,C 180,E1 -21299.161,E2 -21299.161} C_VEL
LIN {X 0,Y 214.323,Z 509.578,A -85,B 0,C 180,E1 -21301.074,E2 -21301.074} C_VEL
LIN {X 0,Y 210.898,Z 517.476,A -85,B 0,C 180,E1 -21303.264,E2 -21303.264} C_VEL
LIN {X 0,Y 207.371,Z 525.225,A -85,B 0,C 180,E1 -21306.002,E2 -21306.002} C_VEL
LIN {X 0,Y 204.504,Z 531.456,A -85,B 0,C 180,E1 -21308.847,E2 -21308.847} C_VEL
LIN {X 0,Y 202.045,Z 536.438,A -85,B 0,C 180,E1 -21311.756,E2 -21311.756} C_VEL
LIN {X 0,Y 200.013,Z 540.311,A -85,B 0,C 180,E1 -21314.72,E2 -21314.72} C_VEL
LIN {X 0,Y 198.644,Z 543.183,A -85,B 0,C 180,E1 -21317.743,E2 -21317.743} C_VEL
LIN {X 0,Y 197.592,Z 545.545,A -85,B 0,C 180,E1 -21321.82,E2 -21321.82} C_VEL
LIN {X 0,Y 197.344,Z 546.15,A -85,B 0,C 180,E1 -21323.866,E2 -21323.866} C_VEL
LIN {X 0,Y 197.253,Z 546.336,A -85,B 0,C 180,E1 -21326.056,E2 -21326.056} C_VEL
LIN {X 0,Y 197.356,Z 546.129,A -85,B 0,C 180,E1 -21327.959,E2 -21327.959} C_VEL
LIN {X 0,Y 197.49,Z 545.526,A -85,B 0,C 180,E1 -21329.999,E2 -21329.999} C_VEL
LIN {X 0,Y 197.372,Z 544.514,A -85,B 0,C 180,E1 -21332.04,E2 -21332.04} C_VEL
LIN {X 0,Y 197.345,Z 542.871,A -85,B 0,C 180,E1 -21334.313,E2 -21334.313} C_VEL
LIN {X 0,Y 197.595,Z 538.822,A -85,B 0,C 180,E1 -21338.178,E2 -21338.178} C_VEL
LIN {X 0,Y 198.136,Z 534.37,A -85,B 0,C 180,E1 -21341.249,E2 -21341.249} C_VEL
LIN {X 0,Y 199.123,Z 528.7,A -85,B 0,C 180,E1 -21344.303,E2 -21344.303} C_VEL
LIN {X 0,Y 200.739,Z 521.602,A -85,B 0,C 180,E1 -21347.312,E2 -21347.312} C_VEL
LIN {X 0,Y 202.437,Z 514.352,A -85,B 0,C 180,E1 -21349.784,E2 -21349.784} C_VEL
LIN {X 0,Y 204.228,Z 505.52,A -85,B 0,C 180,E1 -21352.242,E2 -21352.242} C_VEL
LIN {X 0,Y 206.583,Z 494.666,A -85,B 0,C 180,E1 -21354.628,E2 -21354.628} C_VEL
LIN {X 0,Y 208.785,Z 483.824,A -85,B 0,C 180,E1 -21356.487,E2 -21356.487} C_VEL
LIN {X 0,Y 210.768,Z 472.635,A -85,B 0,C 180,E1 -21357.963,E2 -21357.963} C_VEL
LIN {X 0,Y 212.55,Z 460.185,A -85,B 0,C 180,E1 -21359.189,E2 -21359.189} C_VEL
LIN {X 0,Y 213.934,Z 447.097,A -85,B 0,C 180,E1 -21360.082,E2 -21360.082} C_VEL
LIN {X 0,Y 214.715,Z 431.373,A -85,B 0,C 180,E1 -21360.709,E2 -21360.709} C_VEL
LIN {X 0,Y 216.218,Z 389.677,A -85,B 0,C 180,E1 -21362.041,E2 -21362.041} C_VEL
LIN {X 0,Y 213.193,Z 361.753,A -85,B 0,C 180,E1 -21363.519,E2 -21363.519} C_VEL
LIN {X 0,Y 206.507,Z 344.552,A -85,B 0,C 180,E1 -21365.235,E2 -21365.235} C_VEL
LIN {X 0,Y 201.518,Z 333.15,A -85,B 0,C 180,E1 -21366.572,E2 -21366.572} C_VEL
LIN {X 0,Y 199.663,Z 325.615,A -85,B 0,C 180,E1 -21370.441,E2 -21370.441} C_VEL
LIN {X 0,Y 199.576,Z 325.625,A -85,B 0,C 180,E1 -21375.227,E2 -21375.227} C_VEL
LIN {X 0,Y 199.576,Z 325.626,A -85,B 0,C 180,E1 -21378.003,E2 -21378.003} C_VEL
LIN {X 0,Y 199.609,Z 325.625,A -85,B 0,C 180,E1 -21380.767,E2 -21380.767} C_VEL
LIN {X 0,Y 199.611,Z 325.622,A -85,B 0,C 180,E1 -21385.713,E2 -21385.713} C_VEL
LIN {X 0,Y 199.699,Z 325.61,A -85,B 0,C 180,E1 -21388.136,E2 -21388.136} C_VEL
LIN {X 0,Y 199.685,Z 325.614,A -85,B 0,C 180,E1 -21392.771,E2 -21392.771} C_VEL
LIN {X 0,Y 199.736,Z 325.605,A -85,B 0,C 180,E1 -21397.228,E2 -21397.228} C_VEL
LIN {X 0,Y 199.794,Z 325.595,A -85,B 0,C 180,E1 -21401.757,E2 -21401.757} C_VEL
LIN {X 0,Y 199.834,Z 325.587,A -85,B 0,C 180,E1 -21405.748,E2 -21405.748} C_VEL
LIN {X 0,Y 200.067,Z 325.545,A -85,B 0,C 180,E1 -21409.884,E2 -21409.884} C_VEL
LIN {X 0,Y 200.03,Z 325.568,A -85,B 0,C 180,E1 -21413.949,E2 -21413.949} C_VEL
LIN {X 0,Y 200.318,Z 325.513,A -85,B 0,C 180,E1 -21417.989,E2 -21417.989} C_VEL
LIN {X 0,Y 200.473,Z 325.492,A -85,B 0,C 180,E1 -21420,E2 -21420} C_VEL
LIN {X 0,Y 200.019,Z 325.571,A -85,B 0,C 180,E1 -21424.029,E2 -21424.029} C_VEL
LIN {X 0,Y 200.075,Z 325.547,A -85,B 0,C 180,E1 -21428.077,E2 -21428.077} C_VEL
LIN {X 0,Y 199.871,Z 325.577,A -85,B 0,C 180,E1 -21432.179,E2 -21432.179} C_VEL
LIN {X 0,Y 199.801,Z 325.595,A -85,B 0,C 180,E1 -21436.343,E2 -21436.343} C_VEL
LIN {X 0,Y 199.678,Z 325.59,A -85,B 0,C 180,E1 -21440.607,E2 -21440.607} C_VEL
LIN {X 0,Y 199.661,Z 325.614,A -85,B 0,C 180,E1 -21444.985,E2 -21444.985} C_VEL
LIN {X 0,Y 199.671,Z 325.593,A -85,B 0,C 180,E1 -21449.522,E2 -21449.522} C_VEL
LIN {X 0,Y 199.674,Z 325.602,A -85,B 0,C 180,E1 -21452.358,E2 -21452.358} C_VEL
LIN {X 0,Y 199.619,Z 325.61,A -85,B 0,C 180,E1 -21456.763,E2 -21456.763} C_VEL
LIN {X 0,Y 199.604,Z 325.605,A -85,B 0,C 180,E1 -21459.329,E2 -21459.329} C_VEL
LIN {X 0,Y 199.569,Z 325.623,A -85,B 0,C 180,E1 -21462.31,E2 -21462.31} C_VEL
LIN {X 0,Y 199.572,Z 325.612,A -85,B 0,C 180,E1 -21465.228,E2 -21465.228} C_VEL
LIN {X 0,Y 199.567,Z 325.623,A -85,B 0,C 180,E1 -21468.003,E2 -21468.003} C_VEL
LIN {X 0,Y 199.594,Z 325.617,A -85,B 0,C 180,E1 -21470.773,E2 -21470.773} C_VEL
LIN {X 0,Y 199.61,Z 325.62,A -85,B 0,C 180,E1 -21474.076,E2 -21474.076} C_VEL
LIN {X 0,Y 199.683,Z 325.61,A -85,B 0,C 180,E1 -21478.135,E2 -21478.135} C_VEL
LIN {X 0,Y 199.656,Z 325.608,A -85,B 0,C 180,E1 -21483.356,E2 -21483.356} C_VEL
LIN {X 0,Y 200.719,Z 328.579,A -85,B 0,C 180,E1 -21483.708,E2 -21483.708} C_VEL
LIN {X 0,Y 202.162,Z 330.941,A -85,B 0,C 180,E1 -21484.064,E2 -21484.064} C_VEL
LIN {X 0,Y 209.362,Z 344.433,A -85,B 0,C 180,E1 -21485.814,E2 -21485.814} C_VEL
LIN {X 0,Y 213.686,Z 353.894,A -85,B 0,C 180,E1 -21486.848,E2 -21486.848} C_VEL
LIN {X 0,Y 217.277,Z 364.418,A -85,B 0,C 180,E1 -21487.766,E2 -21487.766} C_VEL
LIN {X 0,Y 214.67,Z 428.495,A -85,B 0,C 180,E1 -21489.833,E2 -21489.833} C_VEL
LIN {X 0,Y 213.659,Z 442.181,A -85,B 0,C 180,E1 -21490.672,E2 -21490.672} C_VEL
LIN {X 0,Y 212.319,Z 454.506,A -85,B 0,C 180,E1 -21491.797,E2 -21491.797} C_VEL
LIN {X 0,Y 210.526,Z 466.35,A -85,B 0,C 180,E1 -21493.267,E2 -21493.267} C_VEL
LIN {X 0,Y 208.331,Z 476.505,A -85,B 0,C 180,E1 -21494.845,E2 -21494.845} C_VEL
LIN {X 0,Y 206.278,Z 486.96,A -85,B 0,C 180,E1 -21496.956,E2 -21496.956} C_VEL
LIN {X 0,Y 204.3,Z 495.534,A -85,B 0,C 180,E1 -21499.095,E2 -21499.095} C_VEL
LIN {X 0,Y 202.494,Z 503.425,A -85,B 0,C 180,E1 -21501.518,E2 -21501.518} C_VEL
LIN {X 0,Y 200.63,Z 511.155,A -85,B 0,C 180,E1 -21504.473,E2 -21504.473} C_VEL
LIN {X 0,Y 199.124,Z 518.244,A -85,B 0,C 180,E1 -21507.978,E2 -21507.978} C_VEL
LIN {X 0,Y 198.159,Z 522.983,A -85,B 0,C 180,E1 -21511.017,E2 -21511.017} C_VEL
LIN {X 0,Y 197.752,Z 526.604,A -85,B 0,C 180,E1 -21514.077,E2 -21514.077} C_VEL
LIN {X 0,Y 197.517,Z 528.487,A -85,B 0,C 180,E1 -21516.128,E2 -21516.128} C_VEL
LIN {X 0,Y 197.262,Z 529.911,A -85,B 0,C 180,E1 -21518.194,E2 -21518.194} C_VEL
LIN {X 0,Y 197.261,Z 531.557,A -85,B 0,C 180,E1 -21522.344,E2 -21522.344} C_VEL
LIN {X 0,Y 197.556,Z 531.781,A -85,B 0,C 180,E1 -21524.42,E2 -21524.42} C_VEL
LIN {X 0,Y 198.011,Z 531.542,A -85,B 0,C 180,E1 -21526.604,E2 -21526.604} C_VEL
LIN {X 0,Y 199.228,Z 529.955,A -85,B 0,C 180,E1 -21530.657,E2 -21530.657} C_VEL
LIN {X 0,Y 200.166,Z 528.507,A -85,B 0,C 180,E1 -21532.72,E2 -21532.72} C_VEL
LIN {X 0,Y 201.945,Z 525.618,A -85,B 0,C 180,E1 -21535.676,E2 -21535.676} C_VEL
LIN {X 0,Y 204.314,Z 521.382,A -85,B 0,C 180,E1 -21538.789,E2 -21538.789} C_VEL
LIN {X 0,Y 207.458,Z 515.241,A -85,B 0,C 180,E1 -21542.123,E2 -21542.123} C_VEL
LIN {X 0,Y 210.97,Z 508.045,A -85,B 0,C 180,E1 -21545.075,E2 -21545.075} C_VEL
LIN {X 0,Y 214.175,Z 500.872,A -85,B 0,C 180,E1 -21547.378,E2 -21547.378} C_VEL
LIN {X 0,Y 217.732,Z 492.096,A -85,B 0,C 180,E1 -21549.618,E2 -21549.618} C_VEL
LIN {X 0,Y 221.475,Z 481.288,A -85,B 0,C 180,E1 -21551.789,E2 -21551.789} C_VEL
LIN {X 0,Y 224.675,Z 470.437,A -85,B 0,C 180,E1 -21553.486,E2 -21553.486} C_VEL
LIN {X 0,Y 227.516,Z 458.37,A -85,B 0,C 180,E1 -21554.929,E2 -21554.929} C_VEL
LIN {X 0,Y 229.687,Z 446.587,A -85,B 0,C 180,E1 -21555.977,E2 -21555.977} C_VEL
LIN {X 0,Y 231.305,Z 433.431,A -85,B 0,C 180,E1 -21556.821,E2 -21556.821} C_VEL
LIN {X 0,Y 232.533,Z 419.347,A -85,B 0,C 180,E1 -21557.295,E2 -21557.295} C_VEL
LIN {X 0,Y 234.588,Z 381.535,A -85,B 0,C 180,E1 -21558.385,E2 -21558.385} C_VEL
LIN {X 0,Y 228.832,Z 369.374,A -85,B 0,C 180,E1 -21560.268,E2 -21560.268} C_VEL
LIN {X 0,Y 224.117,Z 360.665,A -85,B 0,C 180,E1 -21561.876,E2 -21561.876} C_VEL
LIN {X 0,Y 216.538,Z 349.013,A -85,B 0,C 180,E1 -21564.61,E2 -21564.61} C_VEL
LIN {X 0,Y 210.3,Z 340.303,A -85,B 0,C 180,E1 -21567.1,E2 -21567.1} C_VEL
LIN {X 0,Y 207.638,Z 336.732,A -85,B 0,C 180,E1 -21568.245,E2 -21568.245} C_VEL
LIN {X 0,Y 206.77,Z 335.65,A -85,B 0,C 180,E1 -21568.627,E2 -21568.627} C_VEL
LIN {X 0,Y 204.446,Z 332.855,A -85,B 0,C 180,E1 -21569.676,E2 -21569.676} C_VEL
LIN {X 0,Y 203.37,Z 330.99,A -85,B 0,C 180,E1 -21570.214,E2 -21570.214} C_VEL
LIN {X 0,Y 200.996,Z 328.91,A -85,B 0,C 180,E1 -21571.321,E2 -21571.321} C_VEL
LIN {X 0,Y 199.887,Z 326.38,A -85,B 0,C 180,E1 -21571.959,E2 -21571.959} C_VEL
LIN {X 0,Y 199.745,Z 325.587,A -85,B 0,C 180,E1 -21572.119,E2 -21572.119} C_VEL
LIN {X 0,Y 199.715,Z 325.593,A -85,B 0,C 180,E1 -21577.227,E2 -21577.227} C_VEL
LIN {X 0,Y 199.797,Z 325.589,A -85,B 0,C 180,E1 -21581.759,E2 -21581.759} C_VEL
LIN {X 0,Y 199.849,Z 325.583,A -85,B 0,C 180,E1 -21585.75,E2 -21585.75} C_VEL
LIN {X 0,Y 200.077,Z 325.553,A -85,B 0,C 180,E1 -21589.885,E2 -21589.885} C_VEL
LIN {X 0,Y 200.133,Z 325.552,A -85,B 0,C 180,E1 -21591.926,E2 -21591.926} C_VEL
LIN {X 0,Y 200.323,Z 325.518,A -85,B 0,C 180,E1 -21597.99,E2 -21597.99} C_VEL
LIN {X 0,Y 200.478,Z 325.51,A -85,B 0,C 180,E1 -21600,E2 -21600} C_VEL
LIN {X 0,Y 200.032,Z 325.56,A -85,B 0,C 180,E1 -21604.03,E2 -21604.03} C_VEL
LIN {X 0,Y 200.114,Z 325.544,A -85,B 0,C 180,E1 -21608.076,E2 -21608.076} C_VEL
LIN {X 0,Y 199.888,Z 325.571,A -85,B 0,C 180,E1 -21612.179,E2 -21612.179} C_VEL
LIN {X 0,Y 199.806,Z 325.582,A -85,B 0,C 180,E1 -21616.344,E2 -21616.344} C_VEL
LIN {X 0,Y 199.684,Z 325.599,A -85,B 0,C 180,E1 -21620.607,E2 -21620.607} C_VEL
LIN {X 0,Y 199.667,Z 325.603,A -85,B 0,C 180,E1 -21624.986,E2 -21624.986} C_VEL
LIN {X 0,Y 199.667,Z 325.606,A -85,B 0,C 180,E1 -21629.524,E2 -21629.524} C_VEL
LIN {X 0,Y 199.631,Z 325.614,A -85,B 0,C 180,E1 -21633.751,E2 -21633.751} C_VEL
LIN {X 0,Y 199.681,Z 325.92,A -85,B 0,C 180,E1 -21634.274,E2 -21634.274} C_VEL
LIN {X 0,Y 200.615,Z 328.592,A -85,B 0,C 180,E1 -21636.552,E2 -21636.552} C_VEL
LIN {X 0,Y 201.488,Z 331.325,A -85,B 0,C 180,E1 -21638.572,E2 -21638.572} C_VEL
LIN {X 0,Y 204.28,Z 335.715,A -85,B 0,C 180,E1 -21639.964,E2 -21639.964} C_VEL
LIN {X 0,Y 206.041,Z 337.993,A -85,B 0,C 180,E1 -21640.771,E2 -21640.771} C_VEL
LIN {X 0,Y 209.132,Z 342.658,A -85,B 0,C 180,E1 -21642.157,E2 -21642.157} C_VEL
LIN {X 0,Y 213.664,Z 349.959,A -85,B 0,C 180,E1 -21644.071,E2 -21644.071} C_VEL
LIN {X 0,Y 218.847,Z 358.846,A -85,B 0,C 180,E1 -21646.101,E2 -21646.101} C_VEL
LIN {X 0,Y 219.491,Z 360.031,A -85,B 0,C 180,E1 -21646.344,E2 -21646.344} C_VEL
LIN {X 0,Y 221.501,Z 364.652,A -85,B 0,C 180,E1 -21647.131,E2 -21647.131} C_VEL
LIN {X 0,Y 222.838,Z 369.922,A -85,B 0,C 180,E1 -21647.74,E2 -21647.74} C_VEL
LIN {X 0,Y 225.566,Z 384.773,A -85,B 0,C 180,E1 -21649.125,E2 -21649.125} C_VEL
LIN {X 0,Y 226.643,Z 388.254,A -85,B 0,C 180,E1 -21649.549,E2 -21649.549} C_VEL
LIN {X 0,Y 227.851,Z 391.704,A -85,B 0,C 180,E1 -21649.996,E2 -21649.996} C_VEL
LIN {X 0,Y 228.642,Z 398.163,A -85,B 0,C 180,E1 -21650.465,E2 -21650.465} C_VEL
LIN {X 0,Y 225.994,Z 442.026,A -85,B 0,C 180,E1 -21651.783,E2 -21651.783} C_VEL
LIN {X 0,Y 224.262,Z 455.506,A -85,B 0,C 180,E1 -21652.485,E2 -21652.485} C_VEL
LIN {X 0,Y 221.857,Z 467.812,A -85,B 0,C 180,E1 -21653.42,E2 -21653.42} C_VEL
LIN {X 0,Y 218.744,Z 479.712,A -85,B 0,C 180,E1 -21654.667,E2 -21654.667} C_VEL
LIN {X 0,Y 215.324,Z 491.106,A -85,B 0,C 180,E1 -21656.298,E2 -21656.298} C_VEL
LIN {X 0,Y 211.603,Z 501.407,A -85,B 0,C 180,E1 -21658.179,E2 -21658.179} C_VEL
LIN {X 0,Y 208.155,Z 509.845,A -85,B 0,C 180,E1 -21660.131,E2 -21660.131} C_VEL
LIN {X 0,Y 203.947,Z 519.015,A -85,B 0,C 180,E1 -21662.832,E2 -21662.832} C_VEL
LIN {X 0,Y 200.099,Z 526.943,A -85,B 0,C 180,E1 -21665.889,E2 -21665.889} C_VEL
LIN {X 0,Y 196.935,Z 533.257,A -85,B 0,C 180,E1 -21669.091,E2 -21669.091} C_VEL
LIN {X 0,Y 194.502,Z 537.799,A -85,B 0,C 180,E1 -21672.113,E2 -21672.113} C_VEL
LIN {X 0,Y 192.553,Z 541.274,A -85,B 0,C 180,E1 -21675.197,E2 -21675.197} C_VEL
LIN {X 0,Y 191.025,Z 544.376,A -85,B 0,C 180,E1 -21679.399,E2 -21679.399} C_VEL
LIN {X 0,Y 190.281,Z 545.917,A -85,B 0,C 180,E1 -21683.638,E2 -21683.638} C_VEL
LIN {X 0,Y 190.256,Z 545.829,A -85,B 0,C 180,E1 -21687.882,E2 -21687.882} C_VEL
LIN {X 0,Y 190.407,Z 545.203,A -85,B 0,C 180,E1 -21689.999,E2 -21689.999} C_VEL
LIN {X 0,Y 190.274,Z 544.167,A -85,B 0,C 180,E1 -21692.116,E2 -21692.116} C_VEL
LIN {X 0,Y 190.243,Z 542.676,A -85,B 0,C 180,E1 -21694.236,E2 -21694.236} C_VEL
LIN {X 0,Y 190.431,Z 539.631,A -85,B 0,C 180,E1 -21697.421,E2 -21697.421} C_VEL
LIN {X 0,Y 190.884,Z 535.5,A -85,B 0,C 180,E1 -21700.607,E2 -21700.607} C_VEL
LIN {X 0,Y 191.991,Z 529.155,A -85,B 0,C 180,E1 -21704.304,E2 -21704.304} C_VEL
LIN {X 0,Y 193.637,Z 522.249,A -85,B 0,C 180,E1 -21707.422,E2 -21707.422} C_VEL
LIN {X 0,Y 195.374,Z 515.186,A -85,B 0,C 180,E1 -21709.982,E2 -21709.982} C_VEL
LIN {X 0,Y 197.212,Z 506.637,A -85,B 0,C 180,E1 -21712.524,E2 -21712.524} C_VEL
LIN {X 0,Y 199.611,Z 496.071,A -85,B 0,C 180,E1 -21714.992,E2 -21714.992} C_VEL
LIN {X 0,Y 201.855,Z 485.614,A -85,B 0,C 180,E1 -21716.911,E2 -21716.911} C_VEL
LIN {X 0,Y 204.001,Z 474.13,A -85,B 0,C 180,E1 -21718.554,E2 -21718.554} C_VEL
LIN {X 0,Y 205.828,Z 462.277,A -85,B 0,C 180,E1 -21719.816,E2 -21719.816} C_VEL
LIN {X 0,Y 207.337,Z 449.215,A -85,B 0,C 180,E1 -21720.793,E2 -21720.793} C_VEL
LIN {X 0,Y 208.175,Z 436.162,A -85,B 0,C 180,E1 -21721.413,E2 -21721.413} C_VEL
LIN {X 0,Y 209.949,Z 390.746,A -85,B 0,C 180,E1 -21722.895,E2 -21722.895} C_VEL
LIN {X 0,Y 207.215,Z 364.165,A -85,B 0,C 180,E1 -21724.344,E2 -21724.344} C_VEL
LIN {X 0,Y 200.777,Z 347.585,A -85,B 0,C 180,E1 -21726.085,E2 -21726.085} C_VEL
LIN {X 0,Y 195.361,Z 335.619,A -85,B 0,C 180,E1 -21727.577,E2 -21727.577} C_VEL
LIN {X 0,Y 194.174,Z 332.784,A -85,B 0,C 180,E1 -21727.973,E2 -21727.973} C_VEL
LIN {X 0,Y 192.557,Z 326.5,A -85,B 0,C 180,E1 -21731.415,E2 -21731.415} C_VEL
LIN {X 0,Y 192.488,Z 326.508,A -85,B 0,C 180,E1 -21736.904,E2 -21736.904} C_VEL
LIN {X 0,Y 192.549,Z 326.503,A -85,B 0,C 180,E1 -21741.647,E2 -21741.647} C_VEL
LIN {X 0,Y 192.597,Z 326.499,A -85,B 0,C 180,E1 -21746.813,E2 -21746.813} C_VEL
LIN {X 0,Y 192.663,Z 326.486,A -85,B 0,C 180,E1 -21751.691,E2 -21751.691} C_VEL
LIN {X 0,Y 192.704,Z 326.481,A -85,B 0,C 180,E1 -21756.348,E2 -21756.348} C_VEL
LIN {X 0,Y 192.73,Z 326.475,A -85,B 0,C 180,E1 -21761.457,E2 -21761.457} C_VEL
LIN {X 0,Y 192.762,Z 326.471,A -85,B 0,C 180,E1 -21765.213,E2 -21765.213} C_VEL
LIN {X 0,Y 192.978,Z 326.424,A -85,B 0,C 180,E1 -21769.508,E2 -21769.508} C_VEL
LIN {X 0,Y 193.058,Z 326.429,A -85,B 0,C 180,E1 -21771.627,E2 -21771.627} C_VEL
LIN {X 0,Y 193.26,Z 326.392,A -85,B 0,C 180,E1 -21777.915,E2 -21777.915} C_VEL
LIN {X 0,Y 193.437,Z 326.367,A -85,B 0,C 180,E1 -21780,E2 -21780} C_VEL
LIN {X 0,Y 192.964,Z 326.449,A -85,B 0,C 180,E1 -21784.177,E2 -21784.177} C_VEL
LIN {X 0,Y 193.025,Z 326.423,A -85,B 0,C 180,E1 -21788.374,E2 -21788.374} C_VEL
LIN {X 0,Y 192.799,Z 326.462,A -85,B 0,C 180,E1 -21792.633,E2 -21792.633} C_VEL
LIN {X 0,Y 192.754,Z 326.47,A -85,B 0,C 180,E1 -21796.959,E2 -21796.959} C_VEL
LIN {X 0,Y 192.612,Z 326.473,A -85,B 0,C 180,E1 -21801.4,E2 -21801.4} C_VEL
LIN {X 0,Y 192.644,Z 326.486,A -85,B 0,C 180,E1 -21804.213,E2 -21804.213} C_VEL
LIN {X 0,Y 192.646,Z 326.471,A -85,B 0,C 180,E1 -21808.892,E2 -21808.892} C_VEL
LIN {X 0,Y 192.596,Z 326.491,A -85,B 0,C 180,E1 -21813.186,E2 -21813.186} C_VEL
LIN {X 0,Y 192.547,Z 326.482,A -85,B 0,C 180,E1 -21818.352,E2 -21818.352} C_VEL
LIN {X 0,Y 192.486,Z 326.506,A -85,B 0,C 180,E1 -21823.095,E2 -21823.095} C_VEL
LIN {X 0,Y 192.481,Z 326.496,A -85,B 0,C 180,E1 -21826.907,E2 -21826.907} C_VEL
LIN {X 0,Y 192.539,Z 326.491,A -85,B 0,C 180,E1 -21831.647,E2 -21831.647} C_VEL
LIN {X 0,Y 192.592,Z 326.495,A -85,B 0,C 180,E1 -21836.814,E2 -21836.814} C_VEL
LIN {X 0,Y 192.607,Z 326.488,A -85,B 0,C 180,E1 -21842.066,E2 -21842.066} C_VEL
LIN {X 0,Y 193.675,Z 329.419,A -85,B 0,C 180,E1 -21842.419,E2 -21842.419} C_VEL
LIN {X 0,Y 195.06,Z 331.67,A -85,B 0,C 180,E1 -21842.786,E2 -21842.786} C_VEL
LIN {X 0,Y 202.037,Z 344.349,A -85,B 0,C 180,E1 -21844.592,E2 -21844.592} C_VEL
LIN {X 0,Y 207.69,Z 356.319,A -85,B 0,C 180,E1 -21846.014,E2 -21846.014} C_VEL
LIN {X 0,Y 210.893,Z 365.347,A -85,B 0,C 180,E1 -21846.864,E2 -21846.864} C_VEL
LIN {X 0,Y 208.313,Z 429.048,A -85,B 0,C 180,E1 -21848.995,E2 -21848.995} C_VEL
LIN {X 0,Y 207.261,Z 442.635,A -85,B 0,C 180,E1 -21849.857,E2 -21849.857} C_VEL
LIN {X 0,Y 205.764,Z 455.412,A -85,B 0,C 180,E1 -21851.067,E2 -21851.067} C_VEL
LIN {X 0,Y 204.063,Z 466.319,A -85,B 0,C 180,E1 -21852.462,E2 -21852.462} C_VEL
LIN {X 0,Y 201.792,Z 476.527,A -85,B 0,C 180,E1 -21854.082,E2 -21854.082} C_VEL
LIN {X 0,Y 199.641,Z 487.023,A -85,B 0,C 180,E1 -21856.255,E2 -21856.255} C_VEL
LIN {X 0,Y 197.372,Z 496.517,A -85,B 0,C 180,E1 -21858.707,E2 -21858.707} C_VEL
LIN {X 0,Y 195.123,Z 505.639,A -85,B 0,C 180,E1 -21861.717,E2 -21861.717} C_VEL
LIN {X 0,Y 193.291,Z 512.99,A -85,B 0,C 180,E1 -21864.785,E2 -21864.785} C_VEL
LIN {X 0,Y 192.042,Z 518.876,A -85,B 0,C 180,E1 -21867.903,E2 -21867.903} C_VEL
LIN {X 0,Y 191.06,Z 523.538,A -85,B 0,C 180,E1 -21871.055,E2 -21871.055} C_VEL
LIN {X 0,Y 190.643,Z 527.087,A -85,B 0,C 180,E1 -21874.229,E2 -21874.229} C_VEL
LIN {X 0,Y 190.38,Z 528.913,A -85,B 0,C 180,E1 -21876.359,E2 -21876.359} C_VEL
LIN {X 0,Y 190.143,Z 530.295,A -85,B 0,C 180,E1 -21878.503,E2 -21878.503} C_VEL
LIN {X 0,Y 190.097,Z 531.279,A -85,B 0,C 180,E1 -21880.653,E2 -21880.653} C_VEL
LIN {X 0,Y 190.225,Z 531.874,A -85,B 0,C 180,E1 -21882.808,E2 -21882.808} C_VEL
LIN {X 0,Y 190.983,Z 531.83,A -85,B 0,C 180,E1 -21886.909,E2 -21886.909} C_VEL
LIN {X 0,Y 191.598,Z 531.146,A -85,B 0,C 180,E1 -21889.277,E2 -21889.277} C_VEL
LIN {X 0,Y 192.408,Z 530.104,A -85,B 0,C 180,E1 -21891.424,E2 -21891.424} C_VEL
LIN {X 0,Y 194.643,Z 526.82,A -85,B 0,C 180,E1 -21895.488,E2 -21895.488} C_VEL
LIN {X 0,Y 197.066,Z 522.836,A -85,B 0,C 180,E1 -21898.781,E2 -21898.781} C_VEL
LIN {X 0,Y 199.852,Z 517.849,A -85,B 0,C 180,E1 -21901.837,E2 -21901.837} C_VEL
LIN {X 0,Y 203.194,Z 511.529,A -85,B 0,C 180,E1 -21904.799,E2 -21904.799} C_VEL
LIN {X 0,Y 207.026,Z 503.546,A -85,B 0,C 180,E1 -21907.666,E2 -21907.666} C_VEL
LIN {X 0,Y 210.895,Z 494.764,A -85,B 0,C 180,E1 -21910.107,E2 -21910.107} C_VEL
LIN {X 0,Y 214.523,Z 485.302,A -85,B 0,C 180,E1 -21912.191,E2 -21912.191} C_VEL
LIN {X 0,Y 217.716,Z 475.331,A -85,B 0,C 180,E1 -21913.951,E2 -21913.951} C_VEL
LIN {X 0,Y 221.01,Z 463.341,A -85,B 0,C 180,E1 -21915.555,E2 -21915.555} C_VEL
LIN {X 0,Y 223.563,Z 451.185,A -85,B 0,C 180,E1 -21916.797,E2 -21916.797} C_VEL
LIN {X 0,Y 225.504,Z 438.218,A -85,B 0,C 180,E1 -21917.748,E2 -21917.748} C_VEL
LIN {X 0,Y 226.756,Z 426.179,A -85,B 0,C 180,E1 -21918.296,E2 -21918.296} C_VEL
LIN {X 0,Y 229.345,Z 384.006,A -85,B 0,C 180,E1 -21919.509,E2 -21919.509} C_VEL
LIN {X 0,Y 224.014,Z 372.728,A -85,B 0,C 180,E1 -21921.354,E2 -21921.354} C_VEL
LIN {X 0,Y 219.785,Z 364.899,A -85,B 0,C 180,E1 -21922.875,E2 -21922.875} C_VEL
LIN {X 0,Y 212.804,Z 354.064,A -85,B 0,C 180,E1 -21925.53,E2 -21925.53} C_VEL
LIN {X 0,Y 206.999,Z 345.87,A -85,B 0,C 180,E1 -21927.961,E2 -21927.961} C_VEL
LIN {X 0,Y 203.835,Z 341.58,A -85,B 0,C 180,E1 -21929.396,E2 -21929.396} C_VEL
LIN {X 0,Y 201.213,Z 338.125,A -85,B 0,C 180,E1 -21930.654,E2 -21930.654} C_VEL
LIN {X 0,Y 200.35,Z 336.982,A -85,B 0,C 180,E1 -21931.085,E2 -21931.085} C_VEL
LIN {X 0,Y 197.9,Z 334.277,A -85,B 0,C 180,E1 -21932.323,E2 -21932.323} C_VEL
LIN {X 0,Y 196.664,Z 332.026,A -85,B 0,C 180,E1 -21933.038,E2 -21933.038} C_VEL
LIN {X 0,Y 194.231,Z 330.172,A -85,B 0,C 180,E1 -21934.333,E2 -21934.333} C_VEL
LIN {X 0,Y 193.007,Z 327.993,A -85,B 0,C 180,E1 -21935.107,E2 -21935.107} C_VEL
LIN {X 0,Y 192.638,Z 326.476,A -85,B 0,C 180,E1 -21935.455,E2 -21935.455} C_VEL
LIN {X 0,Y 192.732,Z 326.466,A -85,B 0,C 180,E1 -21941.459,E2 -21941.459} C_VEL
LIN {X 0,Y 192.773,Z 326.461,A -85,B 0,C 180,E1 -21945.215,E2 -21945.215} C_VEL
LIN {X 0,Y 193.022,Z 326.43,A -85,B 0,C 180,E1 -21949.511,E2 -21949.511} C_VEL
LIN {X 0,Y 193.005,Z 326.43,A -85,B 0,C 180,E1 -21953.729,E2 -21953.729} C_VEL
LIN {X 0,Y 193.265,Z 326.397,A -85,B 0,C 180,E1 -21957.916,E2 -21957.916} C_VEL
LIN {X 0,Y 193.442,Z 326.386,A -85,B 0,C 180,E1 -21960,E2 -21960} C_VEL
LIN {X 0,Y 192.979,Z 326.44,A -85,B 0,C 180,E1 -21964.177,E2 -21964.177} C_VEL
LIN {X 0,Y 193.064,Z 326.424,A -85,B 0,C 180,E1 -21968.373,E2 -21968.373} C_VEL
